C01810=1059.024,240.008,407.416,172.728,33.763,156.284
C01811=1059.018,239.759,407.444,172.726,33.759,156.283
C01812=1059.012,239.511,407.472,172.723,33.755,156.282
C01813=1059.006,239.263,407.499,172.721,33.752,156.282
C01814=1059.000,239.014,407.528,172.719,33.748,156.281
C01815=1058.993,238.765,407.555,172.717,33.744,156.280
C01816=1058.987,238.517,407.582,172.714,33.740,156.279
C01817=1058.981,238.269,407.610,172.712,33.737,156.279
C01818=1058.975,238.020,407.638,172.709,33.733,156.278
C01819=1058.969,237.772,407.665,172.707,33.729,156.277
C01820=1058.962,237.523,407.692,172.705,33.725,156.276
C01821=1058.956,237.275,407.720,172.703,33.721,156.276
C01822=1058.950,237.027,407.748,172.701,33.718,156.275
C01823=1058.944,236.778,407.775,172.699,33.714,156.274
C01824=1058.938,236.530,407.802,172.696,33.710,156.274
C01825=1058.932,236.297,407.829,172.694,33.707,156.273
C01826=1058.926,236.065,407.854,172.691,33.703,156.272
C01827=1058.920,235.833,407.879,172.689,33.700,156.272
C01828=1058.915,235.599,407.906,172.687,33.696,156.271
C01829=1058.909,235.367,407.931,172.685,33.692,156.270
C01830=1058.903,235.135,407.957,172.683,33.689,156.270
C01831=1058.897,234.902,407.983,172.681,33.685,156.269
C01832=1058.892,234.670,408.008,172.679,33.681,156.268
C01833=1058.885,234.421,408.036,172.677,33.678,156.267
C01834=1058.880,234.173,408.063,172.675,33.674,156.267
C01835=1058.873,233.924,408.090,172.673,33.670,156.266
C01836=1058.867,233.676,408.117,172.671,33.666,156.265
C01837=1058.861,233.427,408.145,172.668,33.663,156.265
C01838=1058.855,233.180,408.173,172.666,33.659,156.264
C01839=1058.849,232.930,408.200,172.664,33.655,156.263
C01840=1058.843,232.683,408.227,172.661,33.651,156.262
C01841=1058.836,232.434,408.254,172.659,33.647,156.262
C01842=1058.830,232.185,408.281,172.657,33.644,156.261
C01843=1058.824,231.937,408.309,172.655,33.639,156.260
C01844=1058.818,231.688,408.335,172.653,33.636,156.259
C01845=1058.811,231.440,408.363,172.651,33.632,156.259
C01846=1058.806,231.192,408.390,172.649,33.629,156.258
C01847=1058.800,230.943,408.418,172.647,33.624,156.257
C01848=1058.794,230.695,408.445,172.644,33.621,156.256
C01849=1058.787,230.445,408.472,172.641,33.617,156.256
C01850=1058.781,230.198,408.499,172.639,33.613,156.255
C01851=1058.775,229.949,408.526,172.637,33.609,156.254
C01852=1058.769,229.701,408.553,172.635,33.605,156.254
C01853=1058.763,229.452,408.580,172.633,33.601,156.253
C01854=1058.757,229.204,408.607,172.631,33.598,156.252
C01855=1058.750,228.954,408.634,172.629,33.594,156.251
C01856=1058.744,228.707,408.661,172.627,33.590,156.251
C01857=1058.737,228.458,408.688,172.625,33.587,156.250
C01858=1058.731,228.210,408.714,172.623,33.582,156.249
C01859=1058.725,227.961,408.742,172.620,33.579,156.248
C01860=1058.719,227.713,408.769,172.617,33.575,156.248
C01861=1058.713,227.464,408.795,172.615,33.571,156.247
C01862=1058.707,227.215,408.822,172.613,33.567,156.246
C01863=1058.700,226.967,408.848,172.611,33.564,156.246
C01864=1058.694,226.719,408.876,172.609,33.560,156.245
C01865=1058.688,226.471,408.903,172.607,33.556,156.244
C01866=1058.681,226.221,408.930,172.605,33.552,156.243
C01867=1058.676,225.973,408.957,172.603,33.548,156.243
C01868=1058.670,225.725,408.983,172.601,33.545,156.242
C01869=1058.663,225.476,409.010,172.599,33.540,156.241
C01870=1058.657,225.228,409.037,172.597,33.537,156.241
C01871=1058.650,224.979,409.064,172.595,33.533,156.240
C01872=1058.645,224.731,409.091,172.592,33.529,156.239
C01873=1058.639,224.483,409.117,172.590,33.525,156.238
C01874=1058.632,224.233,409.144,172.588,33.522,156.238
C01875=1058.626,223.985,409.170,172.586,33.517,156.237
C01876=1058.620,223.737,409.197,172.584,33.514,156.236
C01877=1058.614,223.488,409.224,172.582,33.510,156.235
C01878=1058.608,223.240,409.251,172.580,33.506,156.235
C01879=1058.602,222.991,409.277,172.578,33.502,156.234
C01880=1058.595,222.743,409.304,172.576,33.499,156.233
C01881=1058.590,222.506,409.330,172.574,33.495,156.233
C01882=1058.584,222.270,409.354,172.572,33.491,156.232
C01883=1058.578,222.033,409.380,172.570,33.488,156.231
C01884=1058.572,221.797,409.405,172.568,33.484,156.230
C01885=1058.566,221.561,409.430,172.565,33.480,156.230
C01886=1058.561,221.324,409.456,172.563,33.476,156.229
C01887=1058.555,221.088,409.481,172.561,33.472,156.228
C01888=1058.549,220.852,409.507,172.559,33.469,156.228
C01889=1058.543,220.603,409.532,172.557,33.465,156.227
C01890=1058.537,220.354,409.559,172.555,33.461,156.226
C01891=1058.530,220.106,409.585,172.553,33.458,156.225
C01892=1058.524,219.857,409.612,172.551,33.453,156.225
C01893=1058.517,219.609,409.638,172.549,33.450,156.224
C01894=1058.511,219.360,409.665,172.547,33.446,156.223
C01895=1058.505,219.112,409.691,172.545,33.442,156.222
C01896=1058.499,218.863,409.717,172.543,33.438,156.222
C01897=1058.493,218.614,409.744,172.541,33.435,156.221
C01898=1058.486,218.366,409.770,172.539,33.430,156.220
C01899=1058.481,218.118,409.797,172.537,33.427,156.220
C01900=1058.474,217.868,409.823,172.535,33.423,156.219
C01901=1058.468,217.620,409.849,172.532,33.419,156.218
C01902=1058.462,217.372,409.875,172.530,33.415,156.217
C01903=1058.456,217.124,409.902,172.528,33.411,156.217
C01904=1058.449,216.874,409.928,172.526,33.407,156.216
C01905=1058.443,216.626,409.954,172.524,33.404,156.215
C01906=1058.437,216.378,409.980,172.522,33.400,156.215
C01907=1058.431,216.129,410.007,172.520,33.396,156.214
C01908=1058.424,215.880,410.033,172.519,33.392,156.213
C01909=1058.418,215.632,410.059,172.517,33.388,156.212
C01910=1058.412,215.384,410.085,172.515,33.384,156.212
C01911=1058.406,215.135,410.111,172.513,33.380,156.211
C01912=1058.400,214.887,410.137,172.511,33.376,156.210
C01913=1058.394,214.637,410.164,172.509,33.373,156.209
C01914=1058.387,214.389,410.190,172.507,33.368,156.209
C01915=1058.382,214.141,410.216,172.505,33.365,156.208
C01916=1058.375,213.892,410.242,172.503,33.361,156.207
C01917=1058.370,213.644,410.268,172.500,33.357,156.206
C01918=1058.363,213.395,410.294,172.498,33.353,156.206
C01919=1058.358,213.147,410.320,172.496,33.349,156.205
C01920=1058.350,212.898,410.347,172.494,33.345,156.204
C01921=1058.345,212.649,410.373,172.492,33.341,156.203
C01922=1058.338,212.401,410.399,172.490,33.337,156.203
C01923=1058.333,212.152,410.425,172.488,33.334,156.202
C01924=1058.327,211.904,410.451,172.486,33.329,156.201
C01925=1058.320,211.655,410.476,172.485,33.326,156.200
C01926=1058.314,211.405,410.502,172.483,33.321,156.200
C01927=1058.308,211.157,410.528,172.481,33.318,156.199
C01928=1058.302,210.909,410.554,172.479,33.313,156.198
C01929=1058.296,210.660,410.580,172.477,33.310,156.197
C01930=1058.290,210.412,410.606,172.475,33.306,156.197
C01931=1058.283,210.164,410.632,172.473,33.302,156.196
C01932=1058.277,209.915,410.657,172.471,33.298,156.195
C01933=1058.271,209.666,410.683,172.469,33.294,156.194
C01934=1058.265,209.418,410.709,172.467,33.290,156.194
C01935=1058.258,209.168,410.735,172.465,33.287,156.193
C01936=1058.252,208.920,410.761,172.463,33.282,156.192
C01937=1058.246,208.686,410.785,172.461,33.279,156.192
C01938=1058.241,208.453,410.809,172.459,33.275,156.191
C01939=1058.234,208.219,410.833,172.457,33.271,156.190
C01940=1058.229,207.985,410.857,172.455,33.268,156.190
C01941=1058.223,207.751,410.881,172.454,33.264,156.189
C01942=1058.217,207.517,410.906,172.452,33.260,156.188
C01943=1058.212,207.283,410.930,172.450,33.257,156.187
C01944=1058.206,207.049,410.954,172.448,33.253,156.187
C01945=1058.180,205.999,411.059,172.259,33.165,156.176
C01946=1058.174,205.751,411.084,172.256,33.162,156.175
C01947=1058.169,205.502,411.108,172.254,33.159,156.175
C01948=1058.163,205.253,411.133,172.252,33.156,156.174
C01949=1058.157,205.005,411.157,172.249,33.153,156.173
C01950=1058.151,204.756,411.182,172.247,33.150,156.173
C01951=1058.145,204.507,411.207,172.245,33.147,156.172
C01952=1058.139,204.259,411.232,172.242,33.144,156.172
C01953=1058.133,204.010,411.257,172.240,33.140,156.171
C01954=1058.128,203.761,411.281,172.238,33.138,156.171
C01955=1058.122,203.512,411.306,172.235,33.135,156.170
C01956=1058.116,203.263,411.331,172.233,33.132,156.170
C01957=1058.110,203.015,411.355,172.231,33.128,156.169
C01958=1058.104,202.766,411.379,172.228,33.125,156.169
C01959=1058.098,202.518,411.404,172.225,33.122,156.168
C01960=1058.092,202.268,411.429,172.223,33.120,156.168
C01961=1058.087,202.020,411.453,172.220,33.116,156.167
C01962=1058.081,201.771,411.479,172.218,33.113,156.166
C01963=1058.074,201.522,411.503,172.216,33.110,156.166
C01964=1058.069,201.274,411.527,172.213,33.107,156.165
C01965=1058.062,201.025,411.551,172.211,33.104,156.165
C01966=1058.057,200.777,411.576,172.209,33.101,156.164
C01967=1058.050,200.528,411.600,172.207,33.099,156.164
C01968=1058.044,200.278,411.625,172.204,33.095,156.163
C01969=1058.039,200.030,411.649,172.202,33.093,156.163
C01970=1058.032,199.781,411.673,172.200,33.090,156.162
C01971=1058.026,199.533,411.698,172.197,33.087,156.162
C01972=1058.020,199.284,411.722,172.195,33.084,156.161
C01973=1058.015,199.035,411.746,172.193,33.081,156.161
C01974=1058.008,198.786,411.770,172.190,33.078,156.160
C01975=1058.003,198.538,411.794,172.188,33.075,156.160
C01976=1057.996,198.289,411.818,172.186,33.072,156.159
C01977=1057.991,198.040,411.843,172.184,33.069,156.159
C01978=1057.984,197.792,411.868,172.181,33.066,156.158
C01979=1057.978,197.543,411.892,172.179,33.063,156.158
C01980=1057.973,197.294,411.916,172.177,33.061,156.157
C01981=1057.966,197.045,411.940,172.174,33.057,156.157
C01982=1057.961,196.796,411.965,172.172,33.054,156.156
C01983=1057.955,196.548,411.988,172.170,33.052,156.156
C01984=1057.949,196.299,412.013,172.168,33.048,156.155
C01985=1057.943,196.051,412.036,172.166,33.046,156.155
C01986=1057.937,195.801,412.061,172.164,33.043,156.154
C01987=1057.931,195.553,412.085,172.162,33.040,156.154
C01988=1057.925,195.304,412.109,172.160,33.037,156.153
C01989=1057.919,195.055,412.133,172.157,33.034,156.153
C01990=1057.913,194.806,412.158,172.155,33.031,156.152
C01991=1057.907,194.558,412.181,172.153,33.028,156.152
C01992=1057.901,194.309,412.206,172.151,33.025,156.151
C01993=1057.895,194.060,412.230,172.148,33.022,156.151
C01994=1057.890,193.812,412.254,172.146,33.019,156.150
C01995=1057.883,193.562,412.277,172.144,33.017,156.150
C01996=1057.878,193.314,412.301,172.142,33.014,156.149
C01997=1057.871,193.065,412.325,172.140,33.010,156.149
C01998=1057.866,192.816,412.350,172.137,33.008,156.148
C01999=1057.860,192.568,412.373,172.135,33.005,156.148
C02000=1057.854,192.318,412.398,172.133,33.002,156.147
C02001=1057.848,192.070,412.422,172.131,32.999,156.147
C02002=1057.843,191.821,412.445,172.128,32.996,156.146
C02003=1057.836,191.572,412.469,172.126,32.993,156.146
C02004=1057.831,191.323,412.493,172.124,32.990,156.145
C02005=1057.824,191.074,412.518,172.122,32.987,156.145
C02006=1057.819,190.791,412.544,172.119,32.984,156.144
C02007=1057.812,190.507,412.572,172.117,32.980,156.143
C02008=1057.805,190.223,412.599,172.114,32.977,156.143
C02009=1057.799,189.940,412.627,172.112,32.974,156.142
C02010=1057.792,189.691,412.651,172.110,32.971,156.142
C02011=1057.787,189.442,412.674,172.107,32.968,156.141
C02012=1057.781,189.193,412.698,172.105,32.965,156.141
C02013=1057.774,188.944,412.722,172.103,32.963,156.140
C02014=1057.769,188.695,412.745,172.101,32.959,156.140
C02015=1057.763,188.447,412.769,172.099,32.957,156.139
C02016=1057.758,188.198,412.793,172.096,32.954,156.139
C02017=1057.752,187.949,412.817,172.094,32.951,156.138
C02018=1057.746,187.700,412.841,172.092,32.948,156.138
C02019=1057.740,187.452,412.864,172.090,32.945,156.137
C02020=1057.735,187.203,412.887,172.088,32.942,156.137
C02021=1057.729,186.954,412.912,172.086,32.939,156.136
C02022=1057.723,186.705,412.936,172.083,32.936,156.136
C02023=1057.718,186.456,412.959,172.081,32.933,156.135
C02024=1057.712,186.208,412.983,172.079,32.931,156.135
C02025=1057.706,185.958,413.007,172.077,32.928,156.134
C02026=1057.700,185.710,413.030,172.075,32.925,156.134
C02027=1057.694,185.461,413.054,172.073,32.922,156.133
C02028=1057.689,185.212,413.078,172.071,32.919,156.133
C02029=1057.683,184.964,413.101,172.068,32.916,156.132
C02030=1057.677,184.714,413.125,172.066,32.913,156.132
C02031=1057.671,184.466,413.149,172.064,32.910,156.131
C02032=1057.666,184.217,413.172,172.062,32.908,156.131
C02033=1057.660,183.969,413.196,172.060,32.905,156.130
C02034=1057.653,183.719,413.219,172.058,32.902,156.130
C02035=1057.647,183.470,413.242,172.055,32.899,156.129
C02036=1057.641,183.222,413.265,172.053,32.897,156.129
C02037=1057.635,182.972,413.289,172.051,32.894,156.128
C02038=1057.629,182.724,413.312,172.049,32.891,156.128
C02039=1057.623,182.475,413.335,172.047,32.889,156.128
C02040=1057.618,182.226,413.358,172.045,32.886,156.127
C02041=1057.610,181.977,413.382,172.042,32.883,156.127
C02042=1057.604,181.729,413.405,172.040,32.880,156.126
C02043=1057.599,181.480,413.428,172.038,32.878,156.126
C02044=1057.593,181.231,413.451,172.036,32.875,156.125
C02045=1057.586,180.982,413.475,172.034,32.872,156.125
C02046=1057.581,180.733,413.498,172.032,32.869,156.124
C02047=1057.575,180.485,413.521,172.030,32.867,156.124
C02048=1057.569,180.236,413.544,172.027,32.864,156.123
C02049=1057.563,179.986,413.567,172.025,32.862,156.123
C02050=1057.557,179.737,413.590,172.023,32.858,156.122
C02051=1057.550,179.489,413.613,172.021,32.856,156.122
C02052=1057.544,179.240,413.636,172.019,32.853,156.122
C02053=1057.539,178.991,413.659,172.017,32.851,156.121
C02054=1057.532,178.742,413.683,172.015,32.848,156.121
C02055=1057.526,178.494,413.706,172.013,32.845,156.120
C02056=1057.520,178.245,413.729,172.011,32.842,156.120
C02057=1057.515,177.996,413.752,172.009,32.840,156.119
C02058=1057.509,177.747,413.775,172.007,32.837,156.119
C02059=1057.502,177.498,413.798,172.005,32.834,156.118
C02060=1057.496,177.249,413.822,172.003,32.831,156.118
C02061=1057.490,177.000,413.845,172.001,32.829,156.117
C02062=1057.484,176.752,413.867,171.999,32.826,156.117
C02063=1057.479,176.503,413.890,171.997,32.823,156.116
C02064=1057.473,176.254,413.913,171.995,32.821,156.116
C02065=1057.467,176.005,413.936,171.993,32.818,156.116
C02066=1057.461,175.756,413.959,171.990,32.815,156.115
C02067=1057.454,175.507,413.982,171.988,32.812,156.115
C02068=1057.448,175.258,414.006,171.986,32.810,156.114
C02069=1057.443,175.009,414.029,171.984,32.807,156.114
C02070=1057.436,174.725,414.054,171.982,32.804,156.113
C02071=1057.429,174.441,414.081,171.979,32.801,156.113
C02072=1057.422,174.156,414.107,171.977,32.798,156.112
C02073=1057.416,173.872,414.133,171.975,32.795,156.112
C02074=1057.410,173.623,414.156,171.973,32.792,156.111
C02075=1057.404,173.374,414.178,171.971,32.789,156.111
C02076=1057.398,173.125,414.201,171.968,32.786,156.110
C02077=1057.393,172.876,414.224,171.966,32.784,156.110
C02078=1057.386,172.628,414.247,171.964,32.781,156.109
C02079=1057.380,172.379,414.270,171.962,32.778,156.109
C02080=1057.375,172.130,414.293,171.960,32.776,156.108
C02081=1057.369,171.881,414.316,171.958,32.773,156.108
C02082=1057.363,171.632,414.339,171.956,32.770,156.108
C02083=1057.357,171.384,414.361,171.954,32.768,156.107
C02084=1057.351,171.135,414.384,171.952,32.765,156.107
C02085=1057.345,170.886,414.407,171.950,32.762,156.106
C02086=1057.340,170.637,414.430,171.948,32.760,156.106
C02087=1057.334,170.388,414.453,171.946,32.757,156.105
C02088=1057.327,170.139,414.475,171.944,32.754,156.105
C02089=1057.322,169.891,414.498,171.942,32.751,156.104
C02090=1057.316,169.641,414.520,171.940,32.749,156.104
C02091=1057.311,169.392,414.543,171.939,32.746,156.103
C02092=1057.305,169.143,414.566,171.937,32.744,156.103
C02093=1057.298,168.895,414.588,171.935,32.740,156.102
C02094=1057.293,168.646,414.611,171.933,32.738,156.102
C02095=1057.287,168.397,414.634,171.931,32.735,156.102
C02096=1057.281,168.147,414.657,171.929,32.733,156.101
C02097=1057.275,167.899,414.679,171.927,32.730,156.101
C02098=1057.269,167.650,414.702,171.925,32.727,156.100
C02099=1057.264,167.402,414.724,171.923,32.724,156.100
C02100=1057.258,167.153,414.747,171.921,32.722,156.099
C02101=1057.252,166.904,414.769,171.919,32.719,156.099
C02102=1057.246,166.655,414.792,171.917,32.716,156.098
C02103=1057.241,166.406,414.815,171.915,32.713,156.098
C02104=1057.235,166.157,414.838,171.913,32.711,156.097
C02105=1057.229,165.908,414.859,171.911,32.708,156.097
C02106=1057.223,165.659,414.882,171.909,32.706,156.097
C02107=1057.217,165.410,414.905,171.907,32.702,156.096
C02108=1057.213,165.161,414.927,171.905,32.700,156.096
C02109=1057.206,164.913,414.950,171.903,32.697,156.095
C02110=1057.200,164.664,414.973,171.901,32.695,156.095
C02111=1057.195,164.414,414.995,171.899,32.692,156.094
C02112=1057.189,164.165,415.018,171.897,32.689,156.094
C02113=1057.183,163.917,415.040,171.895,32.686,156.093
C02114=1057.177,163.667,415.062,171.893,32.684,156.093
C02115=1057.172,163.419,415.085,171.891,32.681,156.092
C02116=1057.166,163.170,415.108,171.889,32.678,156.092
C02117=1057.160,162.921,415.129,171.887,32.675,156.091
C02118=1057.155,162.672,415.152,171.885,32.673,156.091
C02119=1057.149,162.422,415.175,171.884,32.670,156.091
C02120=1057.143,162.175,415.197,171.882,32.668,156.090
C02121=1057.138,161.926,415.220,171.880,32.665,156.090
C02122=1057.132,161.676,415.242,171.878,32.662,156.089
C02123=1057.126,161.427,415.265,171.876,32.659,156.089
C02124=1057.120,161.178,415.286,171.874,32.657,156.088
C02125=1057.115,160.930,415.309,171.872,32.654,156.088
C02126=1057.109,160.681,415.331,171.870,32.651,156.087
C02127=1057.103,160.432,415.354,171.868,32.648,156.087
C02128=1057.097,160.182,415.375,171.866,32.646,156.087
C02129=1057.091,159.934,415.397,171.864,32.643,156.086
C02130=1057.085,159.684,415.420,171.862,32.641,156.086
C02131=1057.079,159.435,415.441,171.860,32.638,156.085
C02132=1057.074,159.187,415.464,171.858,32.636,156.085
C02133=1057.068,158.938,415.486,171.856,32.633,156.084
C02134=1057.061,158.653,415.511,171.854,32.630,156.084
C02135=1057.054,158.368,415.536,171.852,32.627,156.083
C02136=1057.047,158.084,415.561,171.849,32.624,156.083
C02137=1057.040,157.799,415.586,171.847,32.621,156.082
C02138=1057.034,157.550,415.609,171.845,32.619,156.082
C02139=1057.029,157.302,415.630,171.843,32.616,156.082
C02140=1057.023,157.052,415.652,171.841,32.614,156.081
C02141=1057.017,156.804,415.675,171.839,32.611,156.081
C02142=1057.011,156.554,415.697,171.837,32.608,156.080
C02143=1057.005,156.305,415.718,171.836,32.606,156.080
C02144=1056.999,156.057,415.741,171.835,32.603,156.079
C02145=1056.993,155.808,415.763,171.833,32.601,156.079
C02146=1056.987,155.559,415.784,171.831,32.598,156.079
C02147=1056.981,155.310,415.807,171.829,32.595,156.078
C02148=1056.976,155.061,415.828,171.827,32.593,156.078
C02149=1056.970,154.812,415.850,171.825,32.590,156.077
C02150=1056.963,154.563,415.872,171.823,32.588,156.077
C02151=1056.958,154.314,415.895,171.821,32.585,156.076
C02152=1056.952,154.065,415.916,171.819,32.583,156.076
C02153=1056.946,153.816,415.938,171.817,32.580,156.076
C02154=1056.940,153.567,415.959,171.815,32.577,156.075
C02155=1056.934,153.318,415.981,171.813,32.575,156.075
C02156=1056.928,153.069,416.004,171.811,32.572,156.074
C02157=1056.922,152.820,416.025,171.809,32.570,156.074
C02158=1056.916,152.571,416.047,171.807,32.567,156.073
C02159=1056.910,152.322,416.068,171.805,32.564,156.073
C02160=1056.904,152.073,416.090,171.804,32.562,156.072
C02161=1056.898,151.824,416.111,171.802,32.559,156.072
C02162=1056.893,151.575,416.133,171.800,32.557,156.072
C02163=1056.887,151.325,416.155,171.798,32.554,156.071
C02164=1056.881,151.078,416.177,171.796,32.552,156.071
C02165=1056.875,150.828,416.199,171.795,32.549,156.070
C02166=1056.869,150.579,416.220,171.793,32.546,156.070
C02167=1056.863,150.331,416.242,171.791,32.544,156.069
C02168=1056.858,150.081,416.264,171.789,32.541,156.069
C02169=1056.851,149.832,416.285,171.787,32.539,156.069
C02170=1056.846,149.583,416.307,171.785,32.536,156.068
C02171=1056.840,149.334,416.328,171.784,32.533,156.068
C02172=1056.833,149.085,416.350,171.782,32.531,156.067
C02173=1056.828,148.836,416.371,171.780,32.528,156.067
C02174=1056.822,148.587,416.393,171.778,32.526,156.066
C02175=1056.816,148.338,416.415,171.776,32.523,156.066
C02176=1056.810,148.090,416.436,171.774,32.521,156.066
C02177=1056.804,147.840,416.457,171.772,32.518,156.065
C02178=1056.798,147.591,416.480,171.770,32.516,156.065
C02179=1056.792,147.343,416.500,171.768,32.513,156.064
C02180=1056.786,147.093,416.522,171.766,32.511,156.064
C02181=1056.780,146.844,416.544,171.765,32.508,156.064
C02182=1056.774,146.596,416.565,171.763,32.506,156.063
C02183=1056.768,146.347,416.587,171.761,32.503,156.063
C02184=1056.762,146.097,416.607,171.759,32.500,156.062
C02185=1056.757,145.848,416.629,171.758,32.498,156.062
C02186=1056.751,145.599,416.650,171.756,32.496,156.062
C02187=1056.744,145.350,416.672,171.754,32.493,156.061
C02188=1056.739,145.101,416.693,171.752,32.491,156.061
C02189=1056.733,144.852,416.715,171.750,32.488,156.060
C02190=1056.726,144.603,416.737,171.748,32.485,156.060
C02191=1056.721,144.354,416.758,171.747,32.483,156.059
C02192=1056.715,144.105,416.779,171.745,32.480,156.059
C02193=1056.709,143.856,416.799,171.743,32.478,156.059
C02194=1056.703,143.607,416.821,171.741,32.476,156.058
C02195=1056.696,143.358,416.843,171.739,32.473,156.058
C02196=1056.691,143.109,416.864,171.737,32.470,156.057
C02197=1056.685,142.860,416.885,171.735,32.468,156.057
C02198=1056.678,142.575,416.910,171.733,32.465,156.056
C02199=1056.672,142.290,416.934,171.731,32.462,156.056
C02200=1056.665,142.005,416.957,171.729,32.459,156.055
C02201=1056.658,141.720,416.982,171.727,32.456,156.055
C02202=1056.653,141.472,417.004,171.725,32.454,156.055
C02203=1056.646,141.222,417.025,171.724,32.451,156.054
C02204=1056.640,140.973,417.046,171.722,32.448,156.054
C02205=1056.634,140.724,417.067,171.720,32.446,156.053
C02206=1056.628,140.475,417.089,171.719,32.444,156.053
C02207=1056.623,140.226,417.109,171.717,32.441,156.053
C02208=1056.617,139.977,417.131,171.715,32.439,156.052
C02209=1056.611,139.728,417.152,171.713,32.436,156.052
C02210=1056.605,139.478,417.173,171.711,32.434,156.051
C02211=1056.599,139.230,417.194,171.709,32.431,156.051
C02212=1056.593,138.981,417.215,171.707,32.428,156.050
C02213=1056.588,138.732,417.236,171.706,32.426,156.050
C02214=1056.581,138.483,417.257,171.704,32.424,156.050
C02215=1056.575,138.234,417.277,171.702,32.421,156.049
C02216=1056.569,137.985,417.299,171.700,32.419,156.049
C02217=1056.563,137.735,417.321,171.698,32.416,156.048
C02218=1056.557,137.487,417.341,171.696,32.413,156.048
C02219=1056.551,137.237,417.362,171.695,32.411,156.048
C02220=1056.546,136.988,417.383,171.693,32.409,156.047
C02221=1056.539,136.739,417.404,171.692,32.406,156.047
C02222=1056.533,136.490,417.424,171.690,32.404,156.046
C02223=1056.527,136.241,417.446,171.688,32.401,156.046
C02224=1056.521,135.992,417.466,171.686,32.398,156.046
C02225=1056.515,135.743,417.488,171.684,32.396,156.045
C02226=1056.510,135.494,417.508,171.683,32.394,156.045
C02227=1056.503,135.245,417.529,171.681,32.391,156.044
C02228=1056.498,134.996,417.550,171.679,32.389,156.044
C02229=1056.492,134.747,417.571,171.677,32.386,156.043
C02230=1056.486,134.498,417.591,171.675,32.384,156.043
C02231=1056.479,134.249,417.613,171.673,32.381,156.043
C02232=1056.474,134.000,417.634,171.672,32.379,156.042
C02233=1056.468,133.751,417.654,171.670,32.376,156.042
C02234=1056.462,133.502,417.675,171.668,32.374,156.041
C02235=1056.457,133.252,417.696,171.666,32.371,156.041
C02236=1056.450,133.004,417.717,171.664,32.369,156.041
C02237=1056.445,132.754,417.737,171.664,32.367,156.040
C02238=1056.438,132.506,417.758,171.662,32.364,156.040
C02239=1056.432,132.256,417.779,171.660,32.361,156.039
C02240=1056.427,132.007,417.799,171.658,32.359,156.039
C02241=1056.420,131.758,417.820,171.656,32.356,156.039
C02242=1056.415,131.509,417.841,171.654,32.354,156.038
C02243=1056.408,131.260,417.861,171.653,32.352,156.038
C02244=1056.403,131.011,417.883,171.651,32.349,156.037
C02245=1056.396,130.762,417.903,171.649,32.347,156.037
C02246=1056.390,130.513,417.923,171.647,32.344,156.037
C02247=1056.384,130.264,417.945,171.645,32.342,156.036
C02248=1056.378,130.015,417.965,171.644,32.340,156.036
C02249=1056.372,129.765,417.985,171.642,32.337,156.035
C02250=1056.366,129.516,418.005,171.640,32.335,156.035
C02251=1056.359,129.267,418.026,171.638,32.332,156.035
C02252=1056.353,129.019,418.046,171.636,32.330,156.034
C02253=1056.348,128.769,418.067,171.635,32.327,156.034
C02254=1056.342,128.520,418.087,171.634,32.325,156.033
C02255=1056.336,128.271,418.109,171.632,32.323,156.033
C02256=1056.329,128.022,418.129,171.630,32.320,156.033
C02257=1056.323,127.773,418.149,171.628,32.318,156.032
C02258=1056.318,127.523,418.170,171.626,32.315,156.032
C02259=1056.312,127.274,418.190,171.625,32.313,156.032
C02260=1056.306,127.026,418.210,171.623,32.311,156.031
C02261=1056.299,126.776,418.231,171.621,32.308,156.031
C02262=1056.292,126.492,418.254,171.619,32.305,156.030
C02263=1056.285,126.207,418.278,171.617,32.303,156.030
C02264=1056.279,125.922,418.301,171.615,32.300,156.029
C02265=1056.272,125.636,418.324,171.613,32.297,156.029
C02266=1056.266,125.388,418.345,171.611,32.295,156.029
C02267=1056.259,125.138,418.365,171.609,32.292,156.028
C02268=1056.254,124.889,418.385,171.608,32.290,156.028
C02269=1056.248,124.640,418.405,171.607,32.287,156.027
C02270=1056.241,124.391,418.426,171.605,32.285,156.027
C02271=1056.236,124.142,418.446,171.603,32.282,156.027
C02272=1056.230,123.893,418.466,171.601,32.280,156.026
C02273=1056.224,123.643,418.487,171.600,32.277,156.026
C02274=1056.218,123.395,418.507,171.598,32.275,156.025
C02275=1056.212,123.145,418.527,171.596,32.273,156.025
C02276=1056.206,122.896,418.547,171.594,32.270,156.025
C02277=1056.200,122.647,418.567,171.592,32.268,156.024
C02278=1056.194,122.398,418.588,171.591,32.265,156.024
C02279=1056.188,122.148,418.608,171.589,32.263,156.023
C02280=1056.182,121.900,418.628,171.587,32.260,156.023
C02281=1056.177,121.651,418.649,171.585,32.258,156.023
C02282=1056.171,121.402,418.669,171.585,32.256,156.022
C02283=1056.164,121.152,418.689,171.583,32.253,156.022
C02284=1056.158,120.903,418.709,171.581,32.250,156.021
C02285=1056.153,120.654,418.730,171.579,32.248,156.021
C02286=1056.146,120.405,418.750,171.577,32.246,156.021
C02287=1056.140,120.156,418.770,171.576,32.243,156.020
C02288=1056.134,119.907,418.790,171.574,32.241,156.020
C02289=1056.129,119.658,418.810,171.572,32.238,156.019
C02290=1056.122,119.408,418.831,171.570,32.236,156.019
C02291=1056.116,119.160,418.851,171.569,32.234,156.019
C02292=1056.111,118.911,418.871,171.567,32.231,156.018
C02293=1056.105,118.662,418.891,171.565,32.228,156.018
C02294=1056.099,118.412,418.910,171.563,32.226,156.017
C02295=1056.093,118.163,418.931,171.562,32.224,156.017
C02296=1056.088,117.914,418.951,171.561,32.221,156.017
C02297=1056.082,117.665,418.971,171.559,32.218,156.016
C02298=1056.076,117.416,418.991,171.557,32.216,156.016
C02299=1056.070,117.167,419.011,171.556,32.214,156.015
C02300=1056.064,116.917,419.032,171.554,32.211,156.015
C02301=1056.058,116.668,419.051,171.552,32.209,156.015
C02302=1056.052,116.419,419.071,171.550,32.206,156.014
C02303=1056.046,116.170,419.091,171.549,32.204,156.014
C02304=1056.041,115.921,419.112,171.547,32.202,156.013
C02305=1056.034,115.672,419.132,171.545,32.199,156.013
C02306=1056.028,115.422,419.151,171.543,32.196,156.013
C02307=1056.022,115.173,419.171,171.542,32.194,156.012
C02308=1056.016,114.925,419.191,171.540,32.192,156.012
C02309=1056.011,114.676,419.212,171.538,32.189,156.011
C02310=1056.006,114.426,419.231,171.538,32.187,156.011
C02311=1056.000,114.177,419.251,171.536,32.184,156.011
C02312=1055.993,113.928,419.271,171.534,32.181,156.010
C02313=1055.987,113.679,419.291,171.532,32.179,156.010
C02314=1055.981,113.430,419.311,171.531,32.177,156.009
C02315=1055.975,113.181,419.330,171.529,32.174,156.009
C02316=1055.969,112.932,419.350,171.527,32.172,156.009
C02317=1055.963,112.682,419.370,171.525,32.169,156.008
C02318=1055.957,112.433,419.390,171.524,32.167,156.008
C02319=1055.951,112.184,419.410,171.522,32.165,156.008
C02320=1055.945,111.935,419.429,171.520,32.162,156.007
C02321=1055.939,111.686,419.449,171.518,32.160,156.007
C02322=1055.933,111.437,419.469,171.517,32.158,156.006
C02323=1055.927,111.187,419.489,171.516,32.155,156.006
C02324=1055.921,110.938,419.509,171.514,32.153,156.006
C02325=1055.915,110.689,419.528,171.512,32.150,156.005
C02326=1055.908,110.404,419.551,171.510,32.147,156.005
C02327=1055.902,110.118,419.574,171.508,32.145,156.004
C02328=1055.895,109.833,419.596,171.506,32.142,156.004
C02329=1055.888,109.548,419.618,171.505,32.139,156.003
C02330=1055.882,109.300,419.637,171.503,32.137,156.003
C02331=1055.876,109.049,419.657,171.501,32.135,156.003
C02332=1055.870,108.801,419.677,171.499,32.132,156.002
C02333=1055.863,108.551,419.696,171.498,32.130,156.002
C02334=1055.857,108.303,419.716,171.496,32.128,156.002
C02335=1055.851,108.053,419.735,171.495,32.125,156.001
C02336=1055.845,107.804,419.755,171.493,32.123,156.001
C02337=1055.840,107.555,419.774,171.492,32.120,156.000
C02338=1055.833,107.305,419.794,171.490,32.118,156.000
C02339=1055.827,107.056,419.813,171.488,32.116,156.000
C02340=1055.821,106.807,419.833,171.486,32.113,155.999
C02341=1055.815,106.558,419.852,171.485,32.111,155.999
C02342=1055.809,106.309,419.872,171.483,32.109,155.998
C02343=1055.803,106.060,419.891,171.481,32.106,155.998
C02344=1055.797,105.811,419.911,171.480,32.103,155.998
C02345=1055.791,105.562,419.930,171.478,32.101,155.997
C02346=1055.785,105.312,419.949,171.476,32.099,155.997
C02347=1055.779,105.064,419.969,171.474,32.096,155.996
C02348=1055.774,104.814,419.989,171.474,32.094,155.996
C02349=1055.767,104.566,420.008,171.472,32.092,155.996
C02350=1055.761,104.316,420.027,171.470,32.089,155.995
C02351=1055.755,104.067,420.046,171.469,32.087,155.995
C02352=1055.749,103.817,420.067,171.467,32.084,155.995
C02353=1055.743,103.568,420.086,171.465,32.082,155.994
C02354=1055.737,103.319,420.105,171.463,32.080,155.994
C02355=1055.731,103.070,420.125,171.462,32.077,155.993
C02356=1055.725,102.821,420.144,171.460,32.075,155.993
C02357=1055.719,102.571,420.163,171.458,32.072,155.993
C02358=1055.713,102.322,420.183,171.457,32.070,155.992
C02359=1055.707,102.073,420.202,171.455,32.067,155.992
C02360=1055.701,101.824,420.221,171.454,32.065,155.992
C02361=1055.695,101.575,420.241,171.453,32.063,155.991
C02362=1055.690,101.325,420.260,171.451,32.060,155.991
C02363=1055.683,101.076,420.279,171.449,32.058,155.990
C02364=1055.678,100.827,420.298,171.447,32.055,155.990
C02365=1055.672,100.578,420.318,171.446,32.053,155.990
C02366=1055.665,100.329,420.337,171.444,32.051,155.989
C02367=1055.659,100.080,420.356,171.442,32.048,155.989
C02368=1055.654,99.830,420.375,171.441,32.046,155.988
C02369=1055.647,99.581,420.394,171.439,32.044,155.988
C02370=1055.641,99.332,420.414,171.437,32.041,155.988
C02371=1055.635,99.083,420.432,171.435,32.039,155.987
C02372=1055.629,98.834,420.452,171.435,32.036,155.987
C02373=1055.623,98.585,420.470,171.433,32.034,155.987
C02374=1055.617,98.335,420.489,171.431,32.032,155.986
C02375=1055.611,98.086,420.508,171.430,32.029,155.986
C02376=1055.605,97.837,420.528,171.428,32.027,155.985
C02377=1055.598,97.588,420.547,171.426,32.025,155.985
C02378=1055.593,97.339,420.566,171.424,32.022,155.985
C02379=1055.586,97.089,420.585,171.423,32.020,155.984
C02380=1055.580,96.840,420.604,171.421,32.018,155.984
C02381=1055.575,96.591,420.623,171.419,32.015,155.984
C02382=1055.568,96.341,420.642,171.418,32.013,155.983
C02383=1055.563,96.092,420.661,171.417,32.011,155.983
C02384=1055.556,95.843,420.680,171.415,32.008,155.982
C02385=1055.551,95.593,420.699,171.414,32.006,155.982
C02386=1055.544,95.344,420.718,171.412,32.004,155.982
C02387=1055.538,95.096,420.738,171.410,32.001,155.981
C02388=1055.532,94.847,420.756,171.408,31.999,155.981
C02389=1055.527,94.598,420.775,171.407,31.996,155.981
C02390=1055.520,94.312,420.796,171.405,31.994,155.980
C02391=1055.512,94.027,420.818,171.403,31.991,155.980
C02392=1055.506,93.742,420.840,171.401,31.988,155.979
C02393=1055.499,93.457,420.861,171.399,31.986,155.979
C02394=1055.493,93.207,420.880,171.398,31.983,155.978
C02395=1055.487,92.958,420.899,171.397,31.981,155.978
C02396=1055.481,92.709,420.917,171.395,31.978,155.978
C02397=1055.475,92.460,420.937,171.393,31.976,155.977
C02398=1055.468,92.211,420.955,171.392,31.973,155.977
C02399=1055.463,91.961,420.975,171.390,31.971,155.977
C02400=1055.456,91.712,420.993,171.388,31.969,155.976
C02401=1055.451,91.463,421.012,171.387,31.967,155.976
C02402=1055.445,91.214,421.031,171.385,31.964,155.975
C02403=1055.439,90.965,421.050,171.383,31.961,155.975
C02404=1055.433,90.716,421.069,171.382,31.959,155.975
C02405=1055.427,90.466,421.088,171.381,31.957,155.974
C02406=1055.421,90.217,421.107,171.379,31.955,155.974
C02407=1055.414,89.967,421.124,171.377,31.952,155.974
C02408=1055.409,89.718,421.144,171.376,31.950,155.973
C02409=1055.402,89.469,421.162,171.374,31.948,155.973
C02410=1055.396,89.220,421.181,171.372,31.945,155.972
C02411=1055.390,88.971,421.199,171.371,31.943,155.972
C02412=1055.384,88.722,421.219,171.369,31.940,155.972
C02413=1055.378,88.472,421.236,171.367,31.938,155.971
C02414=1055.372,88.223,421.255,171.366,31.936,155.971
C02415=1055.365,87.974,421.274,171.364,31.934,155.971
C02416=1055.359,87.725,421.292,171.363,31.931,155.970
C02417=1055.353,87.475,421.312,171.361,31.929,155.970
C02418=1055.347,87.225,421.330,171.360,31.926,155.969
C02419=1055.341,86.977,421.348,171.358,31.924,155.969
C02420=1055.335,86.728,421.367,171.356,31.922,155.969
C02421=1055.329,86.479,421.386,171.355,31.920,155.968
C02422=1055.323,86.229,421.404,171.353,31.917,155.968
C02423=1055.317,85.980,421.422,171.351,31.915,155.968
C02424=1055.310,85.731,421.441,171.350,31.913,155.967
C02425=1055.304,85.482,421.459,171.348,31.910,155.967
C02426=1055.299,85.232,421.478,171.346,31.908,155.967
C02427=1055.293,84.983,421.496,171.346,31.905,155.966
C02428=1055.286,84.734,421.515,171.344,31.903,155.966
C02429=1055.280,84.484,421.533,171.342,31.901,155.965
C02430=1055.274,84.235,421.552,171.341,31.899,155.965
C02431=1055.269,83.986,421.571,171.339,31.896,155.965
C02432=1055.262,83.736,421.589,171.337,31.894,155.964
C02433=1055.256,83.487,421.607,171.336,31.891,155.964
C02434=1055.250,83.238,421.626,171.334,31.889,155.964
C02435=1055.244,82.989,421.643,171.332,31.887,155.963
C02436=1055.238,82.740,421.663,171.331,31.884,155.963
C02437=1055.232,82.491,421.681,171.330,31.882,155.962
C02438=1055.226,82.241,421.699,171.328,31.879,155.962
C02439=1055.219,81.992,421.718,171.327,31.878,155.962
C02440=1055.214,81.743,421.735,171.325,31.875,155.961
C02441=1055.208,81.493,421.755,171.323,31.873,155.961
C02442=1055.202,81.244,421.773,171.321,31.870,155.961
C02443=1055.196,80.994,421.791,171.320,31.868,155.960
C02444=1055.190,80.746,421.810,171.318,31.866,155.960
C02445=1055.184,80.496,421.827,171.316,31.863,155.959
C02446=1055.177,80.247,421.846,171.315,31.861,155.959
C02447=1055.173,79.998,421.864,171.313,31.858,155.959
C02448=1055.166,79.749,421.883,171.312,31.856,155.958
C02449=1055.160,79.499,421.901,171.311,31.854,155.958
C02450=1055.154,79.250,421.920,171.309,31.851,155.958
C02451=1055.148,79.001,421.938,171.307,31.849,155.957
C02452=1055.142,78.752,421.956,171.306,31.846,155.957
C02453=1055.135,78.503,421.974,171.304,31.844,155.957
C02454=1055.129,78.218,421.995,171.302,31.842,155.956
C02455=1055.122,77.932,422.016,171.300,31.839,155.956
C02456=1055.115,77.647,422.037,171.298,31.836,155.955
C02457=1055.108,77.361,422.058,171.297,31.834,155.955
C02458=1055.102,77.112,422.076,171.296,31.831,155.954
C02459=1055.096,76.864,422.093,171.294,31.829,155.954
C02460=1055.089,76.614,422.111,171.292,31.827,155.954
C02461=1055.083,76.364,422.129,171.291,31.825,155.953
C02462=1055.077,76.116,422.148,171.289,31.822,155.953
C02463=1055.071,75.866,422.166,171.287,31.820,155.953
C02464=1055.065,75.617,422.184,171.286,31.817,155.952
C02465=1055.059,75.367,422.202,171.284,31.815,155.952
C02466=1055.053,75.118,422.220,171.282,31.813,155.952
C02467=1055.047,74.869,422.238,171.282,31.811,155.951
C02468=1055.041,74.619,422.256,171.280,31.808,155.951
C02469=1055.035,74.370,422.274,171.278,31.806,155.951
C02470=1055.029,74.121,422.293,171.277,31.803,155.950
C02471=1055.023,73.871,422.310,171.275,31.801,155.950
C02472=1055.017,73.622,422.328,171.273,31.799,155.949
C02473=1055.010,73.373,422.346,171.272,31.797,155.949
C02474=1055.004,73.124,422.364,171.270,31.794,155.949
C02475=1054.998,72.875,422.382,171.268,31.792,155.948
C02476=1054.992,72.626,422.400,171.267,31.789,155.948
C02477=1054.986,72.376,422.418,171.266,31.787,155.948
C02478=1054.980,72.127,422.436,171.264,31.785,155.947
C02479=1054.974,71.877,422.454,171.263,31.783,155.947
C02480=1054.968,71.629,422.472,171.261,31.780,155.947
C02481=1054.962,71.379,422.490,171.259,31.778,155.946
C02482=1054.955,71.129,422.507,171.258,31.776,155.946
C02483=1054.950,70.880,422.525,171.256,31.773,155.945
C02484=1054.943,70.631,422.543,171.254,31.771,155.945
C02485=1054.937,70.381,422.561,171.253,31.769,155.945
C02486=1054.932,70.132,422.579,171.251,31.766,155.944
C02487=1054.926,69.883,422.597,171.250,31.764,155.944
C02488=1054.920,69.634,422.614,171.249,31.762,155.944
C02489=1054.913,69.385,422.632,171.247,31.760,155.943
C02490=1054.907,69.135,422.650,171.245,31.757,155.943
C02491=1054.901,68.886,422.668,171.244,31.755,155.943
C02492=1054.895,68.636,422.686,171.242,31.752,155.942
C02493=1054.889,68.388,422.703,171.240,31.750,155.942
C02494=1054.883,68.138,422.721,171.239,31.748,155.942
C02495=1054.876,67.889,422.739,171.237,31.746,155.941
C02496=1054.870,67.640,422.756,171.236,31.744,155.941
C02497=1054.864,67.390,422.774,171.235,31.741,155.940
C02498=1054.858,67.141,422.792,171.233,31.739,155.940
C02499=1054.852,66.891,422.810,171.231,31.736,155.940
C02500=1054.846,66.642,422.827,171.230,31.734,155.939
C02501=1054.840,66.393,422.845,171.228,31.732,155.939
C02502=1054.834,66.143,422.863,171.226,31.730,155.939
C02503=1054.828,65.895,422.880,171.224,31.727,155.938
C02504=1054.822,65.645,422.898,171.223,31.725,155.938
C02505=1054.816,65.396,422.915,171.221,31.723,155.938
C02506=1054.809,65.146,422.933,171.220,31.720,155.937
C02507=1054.803,64.897,422.950,171.219,31.718,155.937
C02508=1054.797,64.648,422.968,171.217,31.716,155.937
C02509=1054.791,64.398,422.985,171.215,31.714,155.936
C02510=1054.785,64.149,423.003,171.214,31.711,155.936
C02511=1054.779,63.899,423.021,171.212,31.709,155.936
C02512=1054.773,63.651,423.038,171.210,31.707,155.935
C02513=1054.766,63.401,423.055,171.209,31.704,155.935
C02514=1054.760,63.151,423.073,171.207,31.702,155.934
C02515=1054.753,62.903,423.090,171.206,31.700,155.934
C02516=1054.747,62.653,423.108,171.205,31.698,155.934
C02517=1054.741,62.404,423.125,171.203,31.696,155.933
C02518=1054.734,62.118,423.145,171.201,31.693,155.933
C02519=1054.726,61.833,423.165,171.199,31.690,155.933
C02520=1054.720,61.548,423.185,171.197,31.688,155.932
C02521=1054.713,61.263,423.205,171.195,31.685,155.932
C02522=1054.706,61.013,423.222,171.194,31.683,155.932
C02523=1054.700,60.764,423.239,171.192,31.681,155.931
C02524=1054.694,60.514,423.257,171.191,31.679,155.931
C02525=1054.687,60.266,423.274,171.190,31.677,155.931
C02526=1054.681,60.016,423.292,171.188,31.674,155.930
C02527=1054.675,59.767,423.309,171.186,31.672,155.930
C02528=1054.669,59.517,423.327,171.184,31.669,155.929
C02529=1054.663,59.268,423.343,171.183,31.667,155.929
C02530=1054.656,59.019,423.360,171.181,31.665,155.929
C02531=1054.650,58.770,423.378,171.179,31.663,155.928
C02532=1054.644,58.520,423.395,171.178,31.661,155.928
C02533=1054.638,58.271,423.413,171.177,31.659,155.928
C02534=1054.632,58.021,423.429,171.175,31.656,155.927
C02535=1054.625,57.772,423.446,171.174,31.654,155.927
C02536=1054.619,57.523,423.464,171.172,31.652,155.927
C02537=1054.613,57.274,423.481,171.170,31.649,155.926
C02538=1054.607,57.024,423.499,171.169,31.647,155.926
C02539=1054.601,56.775,423.515,171.167,31.645,155.926
C02540=1054.594,56.525,423.533,171.165,31.643,155.925
C02541=1054.588,56.276,423.550,171.164,31.641,155.925
C02542=1054.582,56.027,423.568,171.163,31.639,155.925
C02543=1054.576,55.777,423.584,171.161,31.636,155.924
C02544=1054.570,55.528,423.601,171.160,31.634,155.924
C02545=1054.563,55.279,423.619,171.158,31.631,155.924
C02546=1054.558,55.029,423.636,171.156,31.629,155.923
C02547=1054.551,54.780,423.653,171.154,31.627,155.923
C02548=1054.545,54.531,423.670,171.153,31.625,155.923
C02549=1054.539,54.281,423.687,171.151,31.622,155.922
C02550=1054.533,54.032,423.704,171.149,31.620,155.922
C02551=1054.527,53.783,423.722,171.149,31.618,155.922
C02552=1054.521,53.533,423.738,171.147,31.616,155.921
C02553=1054.515,53.284,423.755,171.145,31.613,155.921
C02554=1054.508,53.035,423.773,171.144,31.611,155.921
C02555=1054.502,52.785,423.789,171.142,31.609,155.920
C02556=1054.496,52.536,423.806,171.140,31.606,155.920
C02557=1054.490,52.287,423.824,171.139,31.604,155.920
C02558=1054.484,52.037,423.841,171.137,31.602,155.919
C02559=1054.478,51.789,423.858,171.136,31.600,155.919
C02560=1054.472,51.538,423.875,171.135,31.598,155.919
C02561=1054.466,51.290,423.892,171.133,31.595,155.918
C02562=1054.459,51.040,423.909,171.131,31.593,155.918
C02563=1054.454,50.790,423.926,171.130,31.591,155.918
C02564=1054.448,50.542,423.943,171.128,31.588,155.917
C02565=1054.441,50.292,423.960,171.126,31.586,155.917
C02566=1054.435,50.043,423.977,171.125,31.584,155.916
C02567=1054.429,49.793,423.993,171.123,31.582,155.916
C02568=1054.423,49.544,424.011,171.122,31.580,155.916
C02569=1054.417,49.294,424.028,171.121,31.577,155.915
C02570=1054.411,49.045,424.045,171.119,31.575,155.915
C02571=1054.405,48.795,424.061,171.117,31.572,155.915
C02572=1054.399,48.546,424.079,171.116,31.570,155.914
C02573=1054.393,48.297,424.095,171.114,31.568,155.914
C02574=1054.387,48.048,424.112,171.112,31.565,155.914
C02575=1054.381,47.798,424.129,171.111,31.564,155.913
C02576=1054.375,47.549,424.146,171.110,31.561,155.913
C02577=1054.369,47.300,424.162,171.108,31.559,155.913
C02578=1054.363,47.050,424.180,171.106,31.557,155.912
C02579=1054.357,46.801,424.197,171.105,31.554,155.912
C02580=1054.351,46.552,424.214,171.103,31.552,155.912
C02581=1054.345,46.303,424.230,171.101,31.549,155.911
C02582=1054.338,46.017,424.250,171.100,31.547,155.911
C02583=1054.332,45.731,424.269,171.098,31.544,155.910
C02584=1054.324,45.445,424.288,171.096,31.542,155.910
C02585=1054.317,45.160,424.308,171.095,31.539,155.910
C02586=1054.311,44.910,424.324,171.093,31.537,155.909
C02587=1054.305,44.661,424.341,171.091,31.535,155.909
C02588=1054.299,44.412,424.358,171.090,31.532,155.909
C02589=1054.294,44.162,424.374,171.088,31.530,155.908
C02590=1054.287,43.913,424.392,171.086,31.528,155.908
C02591=1054.281,43.664,424.408,171.085,31.525,155.908
C02592=1054.275,43.414,424.424,171.083,31.523,155.907
C02593=1054.269,43.165,424.442,171.082,31.520,155.907
C02594=1054.263,42.915,424.458,171.081,31.519,155.907
C02595=1054.257,42.666,424.475,171.079,31.516,155.906
C02596=1054.250,42.417,424.492,171.077,31.514,155.906
C02597=1054.245,42.168,424.508,171.076,31.512,155.906
C02598=1054.238,41.918,424.524,171.074,31.510,155.905
C02599=1054.232,41.668,424.541,171.072,31.508,155.905
C02600=1054.226,41.420,424.558,171.070,31.505,155.905
C02601=1054.220,41.170,424.574,171.070,31.503,155.904
C02602=1054.213,40.920,424.591,171.068,31.501,155.904
C02603=1054.207,40.671,424.607,171.066,31.498,155.904
C02604=1054.201,40.422,424.624,171.065,31.496,155.903
C02605=1054.195,40.173,424.640,171.063,31.494,155.903
C02606=1054.189,39.923,424.657,171.061,31.492,155.903
C02607=1054.183,39.673,424.673,171.060,31.490,155.902
C02608=1054.177,39.424,424.689,171.058,31.487,155.902
C02609=1054.170,39.175,424.706,171.057,31.485,155.902
C02610=1054.164,38.926,424.722,171.056,31.483,155.901
C02611=1054.158,38.676,424.739,171.054,31.481,155.901
C02612=1054.152,38.426,424.755,171.052,31.479,155.901
C02613=1054.146,38.177,424.772,171.050,31.476,155.900
C02614=1054.141,37.927,424.788,171.049,31.474,155.900
C02615=1054.134,37.679,424.805,171.047,31.472,155.900
C02616=1054.128,37.430,424.821,171.045,31.470,155.899
C02617=1054.121,37.180,424.838,171.045,31.467,155.899
C02618=1054.115,36.930,424.854,171.043,31.465,155.899
C02619=1054.109,36.681,424.870,171.041,31.463,155.898
C02620=1054.103,36.432,424.886,171.040,31.461,155.898
C02621=1054.097,36.182,424.903,171.038,31.459,155.898
C02622=1054.090,35.933,424.919,171.036,31.456,155.897
C02623=1054.084,35.683,424.935,171.034,31.454,155.897
C02624=1054.078,35.434,424.951,171.033,31.452,155.897
C02625=1054.072,35.184,424.967,171.032,31.450,155.896
C02626=1054.066,34.935,424.984,171.030,31.448,155.896
C02627=1054.060,34.685,425.000,171.029,31.445,155.896
C02628=1054.053,34.436,425.016,171.027,31.443,155.895
C02629=1054.047,34.187,425.032,171.025,31.441,155.895
C02630=1054.041,33.937,425.049,171.023,31.439,155.895
C02631=1054.035,33.688,425.065,171.022,31.437,155.894
C02632=1054.029,33.439,425.081,171.020,31.435,155.894
C02633=1054.022,33.189,425.097,171.019,31.432,155.894
C02634=1054.016,32.940,425.113,171.018,31.431,155.894
C02635=1054.010,32.690,425.130,171.016,31.428,155.893
C02636=1054.004,32.441,425.146,171.014,31.426,155.893
C02637=1053.998,32.192,425.162,171.012,31.424,155.893
C02638=1053.992,31.942,425.178,171.011,31.422,155.892
C02639=1053.986,31.693,425.194,171.009,31.420,155.892
C02640=1053.980,31.444,425.210,171.007,31.417,155.892
C02641=1053.974,31.194,425.227,171.007,31.415,155.891
C02642=1053.967,30.944,425.243,171.005,31.413,155.891
C02643=1053.960,30.695,425.259,171.003,31.411,155.891
C02644=1053.955,30.446,425.275,171.001,31.409,155.890
C02645=1053.949,30.197,425.291,171.000,31.406,155.890
C02646=1053.942,29.911,425.310,170.998,31.404,155.890
C02647=1053.935,29.626,425.328,170.996,31.401,155.889
C02648=1053.928,29.339,425.346,170.994,31.399,155.889
C02649=1053.921,29.054,425.365,170.993,31.396,155.889
C02650=1053.915,28.804,425.381,170.991,31.394,155.888
C02651=1053.908,28.555,425.397,170.989,31.392,155.888
C02652=1053.902,28.305,425.412,170.988,31.390,155.888
C02653=1053.897,28.056,425.428,170.986,31.388,155.887
C02654=1053.890,27.807,425.444,170.984,31.385,155.887
C02655=1053.884,27.558,425.460,170.983,31.384,155.887
C02656=1053.877,27.309,425.476,170.982,31.381,155.886
C02657=1053.871,27.058,425.492,170.980,31.379,155.886
C02658=1053.865,26.809,425.508,170.978,31.377,155.886
C02659=1053.858,26.560,425.524,170.977,31.375,155.885
C02660=1053.852,26.310,425.540,170.975,31.373,155.885
C02661=1053.847,26.060,425.556,170.973,31.370,155.885
C02662=1053.840,25.811,425.571,170.971,31.368,155.884
C02663=1053.834,25.562,425.588,170.970,31.366,155.884
C02664=1053.827,25.313,425.603,170.969,31.364,155.884
C02665=1053.822,25.063,425.619,170.967,31.362,155.883
C02666=1053.815,24.814,425.634,170.966,31.360,155.883
C02667=1053.809,24.565,425.651,170.964,31.358,155.883
C02668=1053.803,24.315,425.666,170.962,31.355,155.883
C02669=1053.797,24.066,425.682,170.960,31.353,155.882
C02670=1053.791,23.816,425.698,170.959,31.351,155.882
C02671=1053.784,23.567,425.713,170.957,31.349,155.882
C02672=1053.778,23.317,425.729,170.956,31.347,155.881
C02673=1053.772,23.068,425.745,170.954,31.344,155.881
C02674=1053.766,22.818,425.761,170.953,31.343,155.881
C02675=1053.759,22.569,425.776,170.951,31.340,155.880
C02676=1053.754,22.320,425.793,170.949,31.338,155.880
C02677=1053.747,22.070,425.807,170.947,31.336,155.880
C02678=1053.741,21.821,425.824,170.946,31.334,155.880
C02679=1053.736,21.571,425.839,170.944,31.332,155.879
C02680=1053.729,21.322,425.855,170.943,31.329,155.879
C02681=1053.723,21.072,425.871,170.942,31.327,155.879
C02682=1053.717,20.823,425.886,170.940,31.325,155.878
C02683=1053.711,20.573,425.902,170.938,31.323,155.878
C02684=1053.704,20.324,425.917,170.936,31.321,155.878
C02685=1053.698,20.074,425.934,170.935,31.319,155.877
C02686=1053.692,19.825,425.949,170.933,31.317,155.877
C02687=1053.686,19.575,425.965,170.931,31.315,155.877
C02688=1053.679,19.326,425.980,170.930,31.313,155.876
C02689=1053.673,19.077,425.995,170.929,31.311,155.876
C02690=1053.667,18.827,426.012,170.927,31.309,155.876
C02691=1053.660,18.578,426.027,170.925,31.307,155.876
C02692=1053.655,18.328,426.043,170.923,31.304,155.875
C02693=1053.648,18.079,426.058,170.922,31.302,155.875
C02694=1053.641,17.830,426.073,170.920,31.300,155.875
C02695=1053.636,17.580,426.089,170.919,31.298,155.874
C02696=1053.630,17.331,426.104,170.917,31.296,155.874
C02697=1053.624,17.081,426.120,170.916,31.294,155.874
C02698=1053.618,16.832,426.135,170.914,31.292,155.873
C02699=1053.611,16.583,426.150,170.912,31.290,155.873
C02700=1053.605,16.333,426.166,170.910,31.287,155.873
C02701=1053.599,16.084,426.182,170.909,31.285,155.873
C02702=1053.593,15.834,426.197,170.907,31.283,155.872
C02703=1053.587,15.584,426.212,170.906,31.281,155.872
C02704=1053.580,15.335,426.228,170.904,31.279,155.872
C02705=1053.574,15.085,426.243,170.903,31.277,155.871
C02706=1053.568,14.837,426.259,170.901,31.275,155.871
C02707=1053.562,14.587,426.274,170.899,31.273,155.871
C02708=1053.556,14.337,426.289,170.897,31.271,155.871
C02709=1053.550,14.088,426.305,170.895,31.269,155.870
C02710=1053.542,13.781,426.323,170.894,31.266,155.870
C02711=1053.534,13.475,426.342,170.892,31.263,155.869
C02712=1053.526,13.170,426.361,170.890,31.261,155.869
C02713=1053.518,12.863,426.379,170.888,31.258,155.869
C02714=1053.512,12.624,426.394,170.886,31.256,155.868
C02715=1053.507,12.386,426.408,170.884,31.255,155.868
C02716=1053.501,12.147,426.423,170.883,31.253,155.868
C02717=1053.494,11.909,426.438,170.882,31.251,155.868
C02718=1053.489,11.671,426.452,170.880,31.249,155.867
C02719=1053.482,11.432,426.467,170.879,31.247,155.867
C02720=1053.476,11.193,426.481,170.877,31.245,155.867
C02721=1053.470,10.955,426.496,170.875,31.243,155.867
C02722=1053.464,10.705,426.511,170.873,31.241,155.866
C02723=1053.458,10.456,426.526,170.872,31.239,155.866
C02724=1053.452,10.206,426.541,170.870,31.237,155.866
C02725=1053.445,9.957,426.556,170.869,31.235,155.865
C02726=1053.439,9.707,426.571,170.867,31.233,155.865
C02727=1053.433,9.458,426.586,170.865,31.231,155.865
C02728=1053.426,9.208,426.601,170.864,31.229,155.865
C02729=1053.420,8.959,426.616,170.862,31.226,155.864
C02730=1053.415,8.709,426.631,170.860,31.225,155.864
C02731=1053.408,8.460,426.647,170.858,31.223,155.864
C02732=1053.402,8.210,426.662,170.857,31.221,155.864
C02733=1053.395,7.961,426.677,170.856,31.219,155.863
C02734=1053.389,7.711,426.692,170.854,31.217,155.863
C02735=1053.383,7.462,426.707,170.852,31.215,155.863
C02736=1053.377,7.213,426.721,170.850,31.212,155.862
C02737=1053.370,6.963,426.736,170.849,31.210,155.862
C02738=1053.364,6.714,426.752,170.847,31.208,155.862
C02739=1053.358,6.464,426.768,170.845,31.206,155.862
C02740=1053.352,6.215,426.782,170.844,31.204,155.861
C02741=1053.346,5.965,426.797,170.842,31.202,155.861
C02742=1053.339,5.716,426.812,170.841,31.200,155.861
C02743=1053.333,5.466,426.827,170.839,31.198,155.860
C02744=1053.327,5.217,426.842,170.837,31.196,155.860
C02745=1053.321,4.967,426.857,170.835,31.194,155.860
C02746=1053.314,4.718,426.871,170.834,31.192,155.860
C02747=1053.308,4.468,426.886,170.833,31.190,155.859
C02748=1053.302,4.219,426.901,170.831,31.188,155.859
C02749=1053.296,3.969,426.916,170.829,31.186,155.859
C02750=1053.290,3.719,426.932,170.827,31.184,155.858
C02751=1053.284,3.470,426.946,170.826,31.182,155.858
C02752=1053.278,3.221,426.961,170.824,31.180,155.858
C02753=1053.272,2.971,426.976,170.822,31.178,155.858
C02754=1053.265,2.722,426.991,170.820,31.176,155.857
C02755=1053.260,2.473,427.006,170.819,31.174,155.857
C02756=1053.253,2.223,427.020,170.818,31.172,155.857
C02757=1053.247,1.973,427.035,170.816,31.170,155.857
C02758=1053.240,1.724,427.050,170.814,31.168,155.856
C02759=1053.235,1.475,427.065,170.812,31.166,155.856
C02760=1053.228,1.225,427.080,170.810,31.164,155.856
C02761=1053.222,0.975,427.095,170.809,31.162,155.855
C02762=1053.216,0.726,427.109,170.808,31.159,155.855
C02763=1053.210,0.477,427.124,170.806,31.157,155.855
C02764=1053.203,0.227,427.139,170.804,31.155,155.854
C02765=1053.198,-0.022,427.154,170.802,31.153,155.854
C02766=1053.191,-0.272,427.168,170.801,31.152,155.854
C02767=1053.185,-0.522,427.183,170.799,31.150,155.854
C02768=1053.180,-0.771,427.198,170.797,31.147,155.853
C02769=1053.174,-1.021,427.213,170.796,31.145,155.853
C02770=1053.168,-1.270,427.228,170.794,31.143,155.853
C02771=1053.162,-1.519,427.243,170.793,31.141,155.853
C02772=1053.155,-1.769,427.258,170.791,31.139,155.852
C02773=1053.149,-2.018,427.272,170.789,31.137,155.852
C02774=1053.142,-2.301,427.289,170.787,31.135,155.852
C02775=1053.135,-2.584,427.305,170.785,31.133,155.851
C02776=1053.129,-2.866,427.322,170.784,31.130,155.851
C02777=1053.122,-3.148,427.339,170.782,31.128,155.851
C02778=1053.116,-3.398,427.353,170.780,31.126,155.850
C02779=1053.109,-3.648,427.367,170.778,31.124,155.850
C02780=1053.103,-3.896,427.382,170.776,31.122,155.850
C02781=1053.097,-4.146,427.397,170.774,31.120,155.850
C02782=1053.090,-4.396,427.411,170.773,31.118,155.849
C02783=1053.084,-4.645,427.425,170.772,31.117,155.849
C02784=1053.078,-4.895,427.440,170.770,31.114,155.849
C02785=1053.071,-5.144,427.455,170.768,31.112,155.849
C02786=1053.066,-5.394,427.469,170.766,31.110,155.848
C02787=1053.059,-5.643,427.483,170.764,31.109,155.848
C02788=1053.052,-5.893,427.498,170.763,31.107,155.848
C02789=1053.047,-6.143,427.512,170.761,31.105,155.848
C02790=1053.040,-6.392,427.526,170.759,31.103,155.847
C02791=1053.034,-6.641,427.541,170.758,31.101,155.847
C02792=1053.028,-6.891,427.555,170.756,31.099,155.847
C02793=1053.021,-7.141,427.570,170.754,31.097,155.847
C02794=1053.015,-7.389,427.584,170.752,31.095,155.846
C02795=1053.009,-7.640,427.598,170.751,31.093,155.846
C02796=1053.003,-7.889,427.613,170.749,31.091,155.846
C02797=1052.996,-8.139,427.626,170.747,31.090,155.846
C02798=1052.990,-8.388,427.641,170.746,31.087,155.845
C02799=1052.984,-8.637,427.656,170.744,31.085,155.845
C02800=1052.978,-8.887,427.670,170.742,31.083,155.845
C02801=1052.971,-9.136,427.684,170.741,31.082,155.845
C02802=1052.965,-9.386,427.698,170.739,31.080,155.844
C02803=1052.960,-9.635,427.713,170.737,31.078,155.844
C02804=1052.952,-9.885,427.727,170.735,31.076,155.844
C02805=1052.947,-10.134,427.741,170.734,31.074,155.844
C02806=1052.941,-10.384,427.756,170.732,31.072,155.843
C02807=1052.934,-10.634,427.770,170.730,31.070,155.843
C02808=1052.928,-10.883,427.784,170.729,31.068,155.843
C02809=1052.922,-11.133,427.799,170.727,31.066,155.843
C02810=1052.915,-11.382,427.813,170.725,31.064,155.842
C02811=1052.909,-11.632,427.827,170.723,31.063,155.842
C02812=1052.904,-11.881,427.841,170.722,31.060,155.842
C02813=1052.897,-12.131,427.856,170.720,31.058,155.842
C02814=1052.891,-12.380,427.870,170.718,31.057,155.841
C02815=1052.885,-12.630,427.884,170.717,31.055,155.841
C02816=1052.879,-12.879,427.898,170.715,31.053,155.841
C02817=1052.872,-13.129,427.912,170.713,31.051,155.841
C02818=1052.866,-13.378,427.927,170.711,31.049,155.840
C02819=1052.860,-13.628,427.941,170.710,31.047,155.840
C02820=1052.854,-13.878,427.954,170.708,31.045,155.840
C02821=1052.848,-14.127,427.969,170.706,31.043,155.840
C02822=1052.842,-14.377,427.982,170.705,31.041,155.839
C02823=1052.836,-14.625,427.997,170.703,31.040,155.839
C02824=1052.830,-14.876,428.011,170.701,31.038,155.839
C02825=1052.823,-15.124,428.025,170.699,31.035,155.839
C02826=1052.817,-15.375,428.039,170.697,31.034,155.838
C02827=1052.811,-15.624,428.053,170.696,31.032,155.838
C02828=1052.805,-15.874,428.068,170.694,31.030,155.838
C02829=1052.798,-16.123,428.081,170.692,31.028,155.838
C02830=1052.792,-16.373,428.095,170.691,31.026,155.837
C02831=1052.786,-16.622,428.109,170.689,31.025,155.837
C02832=1052.780,-16.872,428.123,170.687,31.022,155.837
C02833=1052.773,-17.121,428.137,170.685,31.021,155.837
C02834=1052.766,-17.371,428.151,170.684,31.019,155.837
C02835=1052.761,-17.620,428.165,170.682,31.017,155.836
C02836=1052.754,-17.870,428.178,170.680,31.015,155.836
C02837=1052.749,-18.120,428.192,170.678,31.014,155.836
C02838=1052.741,-18.400,428.208,170.676,31.012,155.836
C02839=1052.734,-18.681,428.224,170.674,31.009,155.835
C02840=1052.727,-18.962,428.240,170.672,31.007,155.835
C02841=1052.720,-19.243,428.255,170.671,31.005,155.835
C02842=1052.714,-19.493,428.269,170.669,31.004,155.835
C02843=1052.708,-19.742,428.283,170.667,31.001,155.834
C02844=1052.701,-19.991,428.297,170.665,31.000,155.834
C02845=1052.695,-20.241,428.310,170.663,30.998,155.834
C02846=1052.689,-20.490,428.324,170.661,30.996,155.834
C02847=1052.682,-20.740,428.338,170.659,30.994,155.833
C02848=1052.677,-20.990,428.352,170.659,30.993,155.833
C02849=1052.670,-21.239,428.366,170.657,30.991,155.833
C02850=1052.664,-21.488,428.379,170.655,30.989,155.833
C02851=1052.658,-21.738,428.393,170.653,30.987,155.833
C02852=1052.651,-21.988,428.407,170.651,30.985,155.832
C02853=1052.646,-22.238,428.420,170.649,30.983,155.832
C02854=1052.640,-22.487,428.434,170.647,30.982,155.832
C02855=1052.633,-22.737,428.447,170.646,30.980,155.832
C02856=1052.627,-22.986,428.462,170.644,30.978,155.831
C02857=1052.620,-23.236,428.476,170.642,30.976,155.831
C02858=1052.614,-23.485,428.489,170.641,30.975,155.831
C02859=1052.609,-23.735,428.503,170.639,30.972,155.831
C02860=1052.602,-23.985,428.516,170.637,30.971,155.831
C02861=1052.596,-24.234,428.530,170.635,30.969,155.830
C02862=1052.590,-24.483,428.544,170.634,30.967,155.830
C02863=1052.583,-24.733,428.557,170.632,30.965,155.830
C02864=1052.578,-24.983,428.571,170.630,30.964,155.830
C02865=1052.572,-25.232,428.584,170.628,30.961,155.829
C02866=1052.565,-25.481,428.598,170.626,30.960,155.829
C02867=1052.559,-25.732,428.612,170.624,30.958,155.829
C02868=1052.553,-25.980,428.626,170.622,30.956,155.829
C02869=1052.547,-26.230,428.639,170.622,30.954,155.828
C02870=1052.540,-26.480,428.653,170.620,30.953,155.828
C02871=1052.534,-26.729,428.667,170.618,30.951,155.828
C02872=1052.528,-26.978,428.680,170.616,30.949,155.828
C02873=1052.522,-27.229,428.693,170.614,30.948,155.828
C02874=1052.516,-27.479,428.707,170.612,30.945,155.827
C02875=1052.510,-27.728,428.720,170.610,30.944,155.827
C02876=1052.503,-27.978,428.733,170.608,30.942,155.827
C02877=1052.497,-28.227,428.747,170.607,30.940,155.827
C02878=1052.491,-28.476,428.760,170.605,30.939,155.827
C02879=1052.484,-28.726,428.773,170.603,30.937,155.826
C02880=1052.478,-28.976,428.787,170.601,30.935,155.826
C02881=1052.472,-29.225,428.801,170.599,30.934,155.826
C02882=1052.466,-29.474,428.814,170.597,30.932,155.826
C02883=1052.459,-29.724,428.828,170.595,30.930,155.826
C02884=1052.453,-29.974,428.841,170.595,30.928,155.825
C02885=1052.447,-30.223,428.854,170.593,30.927,155.825
C02886=1052.441,-30.473,428.867,170.591,30.925,155.825
C02887=1052.434,-30.723,428.880,170.589,30.923,155.825
C02888=1052.428,-30.972,428.894,170.587,30.922,155.825
C02889=1052.421,-31.221,428.907,170.585,30.920,155.824
C02890=1052.416,-31.471,428.921,170.583,30.918,155.824
C02891=1052.409,-31.721,428.934,170.582,30.917,155.824
C02892=1052.403,-31.971,428.947,170.580,30.915,155.824
C02893=1052.397,-32.220,428.960,170.578,30.913,155.824
C02894=1052.391,-32.469,428.974,170.576,30.911,155.823
C02895=1052.384,-32.719,428.987,170.574,30.910,155.823
C02896=1052.378,-32.968,429.000,170.572,30.908,155.823
C02897=1052.372,-33.218,429.013,170.570,30.906,155.823
C02898=1052.366,-33.468,429.026,170.568,30.905,155.823
C02899=1052.359,-33.717,429.040,170.567,30.903,155.822
C02900=1052.353,-33.967,429.053,170.565,30.901,155.822
C02901=1052.347,-34.217,429.066,170.563,30.899,155.822
C02902=1052.340,-34.497,429.081,170.561,30.897,155.822
C02903=1052.333,-34.777,429.096,170.559,30.896,155.822
C02904=1052.326,-35.057,429.111,170.557,30.894,155.821
C02905=1052.319,-35.337,429.125,170.555,30.892,155.821
C02906=1052.313,-35.587,429.139,170.554,30.890,155.821
C02907=1052.307,-35.836,429.152,170.552,30.888,155.821
C02908=1052.301,-36.086,429.165,170.550,30.887,155.821
C02909=1052.295,-36.335,429.178,170.548,30.885,155.820
C02910=1052.288,-36.584,429.191,170.546,30.883,155.820
C02911=1052.283,-36.834,429.204,170.544,30.882,155.820
C02912=1052.276,-37.084,429.217,170.542,30.880,155.820
C02913=1052.270,-37.333,429.231,170.541,30.879,155.820
C02914=1052.264,-37.583,429.243,170.539,30.876,155.819
C02915=1052.258,-37.833,429.257,170.537,30.875,155.819
C02916=1052.252,-38.082,429.270,170.535,30.873,155.819
C02917=1052.246,-38.332,429.283,170.533,30.872,155.819
C02918=1052.240,-38.581,429.296,170.531,30.870,155.819
C02919=1052.234,-38.831,429.309,170.529,30.868,155.818
C02920=1052.226,-39.081,429.322,170.528,30.867,155.818
C02921=1052.220,-39.330,429.335,170.526,30.865,155.818
C02922=1052.214,-39.580,429.347,170.524,30.863,155.818
C02923=1052.208,-39.829,429.361,170.522,30.862,155.818
C02924=1052.202,-40.079,429.373,170.520,30.860,155.818
C02925=1052.196,-40.328,429.387,170.518,30.859,155.817
C02926=1052.189,-40.578,429.399,170.516,30.857,155.817
C02927=1052.183,-40.827,429.412,170.515,30.856,155.817
C02928=1052.176,-41.078,429.425,170.513,30.854,155.817
C02929=1052.170,-41.327,429.438,170.511,30.852,155.817
C02930=1052.164,-41.577,429.451,170.509,30.851,155.816
C02931=1052.157,-41.826,429.463,170.507,30.849,155.816
C02932=1052.152,-42.076,429.476,170.505,30.848,155.816
C02933=1052.145,-42.325,429.489,170.503,30.846,155.816
C02934=1052.139,-42.575,429.502,170.501,30.844,155.816
C02935=1052.133,-42.824,429.515,170.500,30.843,155.816
C02936=1052.127,-43.074,429.527,170.498,30.841,155.815
C02937=1052.120,-43.323,429.540,170.496,30.840,155.815
C02938=1052.114,-43.573,429.553,170.494,30.838,155.815
C02939=1052.108,-43.823,429.565,170.492,30.837,155.815
C02940=1052.102,-44.072,429.578,170.490,30.835,155.815
C02941=1052.095,-44.322,429.591,170.488,30.834,155.815
C02942=1052.089,-44.572,429.604,170.487,30.832,155.815
C02943=1052.083,-44.821,429.617,170.485,30.830,155.814
C02944=1052.077,-45.071,429.629,170.483,30.828,155.814
C02945=1052.071,-45.321,429.642,170.481,30.827,155.814
C02946=1052.064,-45.570,429.654,170.479,30.825,155.814
C02947=1052.058,-45.819,429.668,170.477,30.824,155.814
C02948=1052.052,-46.069,429.680,170.475,30.822,155.813
C02949=1052.046,-46.319,429.693,170.473,30.821,155.813
C02950=1052.040,-46.568,429.706,170.472,30.819,155.813
C02951=1052.033,-46.818,429.718,170.470,30.818,155.813
C02952=1052.027,-47.068,429.731,170.468,30.816,155.813
C02953=1052.021,-47.317,429.744,170.466,30.815,155.813
C02954=1052.015,-47.567,429.756,170.464,30.813,155.812
C02955=1052.009,-47.817,429.768,170.462,30.812,155.812
C02956=1052.003,-48.067,429.781,170.460,30.810,155.812
C02957=1051.996,-48.316,429.794,170.459,30.808,155.812
C02958=1051.991,-48.565,429.806,170.457,30.807,155.812
C02959=1051.984,-48.815,429.818,170.455,30.805,155.812
C02960=1051.979,-49.064,429.831,170.453,30.804,155.811
C02961=1051.972,-49.314,429.844,170.451,30.802,155.811
C02962=1051.966,-49.564,429.857,170.449,30.801,155.811
C02963=1051.960,-49.813,429.869,170.447,30.799,155.811
C02964=1051.954,-50.063,429.881,170.445,30.798,155.811
C02965=1051.948,-50.312,429.894,170.444,30.796,155.811
C02966=1051.940,-50.593,429.908,170.442,30.795,155.810
C02967=1051.933,-50.873,429.922,170.440,30.793,155.810
C02968=1051.926,-51.154,429.935,170.437,30.791,155.810
C02969=1051.919,-51.435,429.950,170.435,30.790,155.810
C02970=1051.913,-51.684,429.961,170.433,30.788,155.810
C02971=1051.907,-51.934,429.974,170.431,30.787,155.810
C02972=1051.900,-52.184,429.986,170.430,30.786,155.810
C02973=1051.894,-52.433,429.999,170.428,30.784,155.810
C02974=1051.887,-52.682,430.011,170.426,30.783,155.809
C02975=1051.880,-52.932,430.023,170.424,30.782,155.809
C02976=1051.875,-53.182,430.036,170.422,30.780,155.809
C02977=1051.868,-53.431,430.048,170.420,30.779,155.809
C02978=1051.862,-53.681,430.060,170.418,30.777,155.809
C02979=1051.855,-53.931,430.072,170.416,30.776,155.809
C02980=1051.849,-54.181,430.085,170.414,30.774,155.809
C02981=1051.843,-54.430,430.097,170.412,30.773,155.808
C02982=1051.836,-54.680,430.109,170.410,30.771,155.808
C02983=1051.831,-54.929,430.121,170.408,30.770,155.808
C02984=1051.824,-55.179,430.133,170.406,30.769,155.808
C02985=1051.818,-55.429,430.145,170.404,30.767,155.808
C02986=1051.812,-55.678,430.157,170.402,30.766,155.808
C02987=1051.805,-55.928,430.169,170.400,30.765,155.808
C02988=1051.799,-56.178,430.182,170.399,30.763,155.808
C02989=1051.792,-56.427,430.194,170.397,30.762,155.807
C02990=1051.786,-56.677,430.206,170.395,30.761,155.807
C02991=1051.780,-56.927,430.218,170.393,30.759,155.807
C02992=1051.773,-57.176,430.230,170.391,30.758,155.807
C02993=1051.768,-57.425,430.242,170.389,30.756,155.807
C02994=1051.761,-57.675,430.254,170.387,30.755,155.807
C02995=1051.755,-57.924,430.266,170.385,30.754,155.807
C02996=1051.749,-58.174,430.279,170.384,30.752,155.806
C02997=1051.742,-58.424,430.291,170.381,30.751,155.806
C02998=1051.735,-58.673,430.303,170.379,30.750,155.806
C02999=1051.730,-58.923,430.315,170.377,30.748,155.806
C03000=1051.724,-59.172,430.327,170.375,30.747,155.806
C03001=1051.718,-59.423,430.339,170.373,30.746,155.806
C03002=1051.711,-59.672,430.351,170.371,30.744,155.806
C03003=1051.705,-59.922,430.363,170.369,30.743,155.806
C03004=1051.699,-60.172,430.375,170.368,30.742,155.806
C03005=1051.693,-60.421,430.387,170.366,30.740,155.805
C03006=1051.686,-60.670,430.399,170.364,30.739,155.805
C03007=1051.680,-60.920,430.411,170.362,30.738,155.805
C03008=1051.674,-61.170,430.423,170.360,30.736,155.805
C03009=1051.667,-61.420,430.435,170.358,30.735,155.805
C03010=1051.662,-61.669,430.447,170.356,30.733,155.805
C03011=1051.655,-61.919,430.459,170.354,30.732,155.805
C03012=1051.649,-62.168,430.471,170.352,30.731,155.805
C03013=1051.643,-62.418,430.483,170.350,30.729,155.804
C03014=1051.637,-62.668,430.494,170.348,30.728,155.804
C03015=1051.630,-62.917,430.506,170.346,30.727,155.804
C03016=1051.624,-63.167,430.519,170.344,30.725,155.804
C03017=1051.618,-63.417,430.531,170.342,30.724,155.804
C03018=1051.612,-63.666,430.542,170.340,30.723,155.804
C03019=1051.606,-63.916,430.554,170.339,30.721,155.804
C03020=1051.599,-64.166,430.566,170.337,30.720,155.804
C03021=1051.593,-64.415,430.578,170.335,30.719,155.804
C03022=1051.587,-64.665,430.589,170.333,30.718,155.803
C03023=1051.581,-64.914,430.601,170.331,30.716,155.803
C03024=1051.574,-65.164,430.613,170.329,30.715,155.803
C03025=1051.569,-65.414,430.624,170.326,30.714,155.803
C03026=1051.563,-65.663,430.637,170.324,30.712,155.803
C03027=1051.556,-65.913,430.649,170.322,30.711,155.803
C03028=1051.550,-66.162,430.660,170.321,30.710,155.803
C03029=1051.544,-66.412,430.672,170.319,30.709,155.803
C03030=1051.537,-66.694,430.685,170.317,30.707,155.803
C03031=1051.530,-66.975,430.699,170.314,30.705,155.802
C03032=1051.523,-67.257,430.712,170.312,30.704,155.802
C03033=1051.516,-67.540,430.725,170.310,30.702,155.802
C03034=1051.510,-67.789,430.737,170.308,30.701,155.802
C03035=1051.504,-68.039,430.749,170.307,30.700,155.802
C03036=1051.498,-68.288,430.760,170.305,30.699,155.802
C03037=1051.492,-68.538,430.772,170.302,30.697,155.802
C03038=1051.486,-68.788,430.784,170.300,30.696,155.802
C03039=1051.480,-69.037,430.795,170.298,30.695,155.802
C03040=1051.473,-69.287,430.806,170.296,30.694,155.801
C03041=1051.467,-69.537,430.819,170.294,30.692,155.801
C03042=1051.461,-69.786,430.831,170.292,30.691,155.801
C03043=1051.455,-70.036,430.842,170.291,30.690,155.801
C03044=1051.449,-70.285,430.853,170.289,30.689,155.801
C03045=1051.443,-70.536,430.865,170.287,30.687,155.801
C03046=1051.437,-70.785,430.877,170.285,30.686,155.801
C03047=1051.431,-71.035,430.888,170.283,30.685,155.801
C03048=1051.424,-71.284,430.900,170.280,30.684,155.801
C03049=1051.419,-71.534,430.912,170.278,30.682,155.801
C03050=1051.413,-71.784,430.924,170.276,30.681,155.800
C03051=1051.407,-72.033,430.934,170.275,30.680,155.800
C03052=1051.400,-72.283,430.946,170.273,30.679,155.800
C03053=1051.395,-72.533,430.958,170.271,30.677,155.800
C03054=1051.389,-72.782,430.970,170.269,30.676,155.800
C03055=1051.382,-73.032,430.981,170.267,30.675,155.800
C03056=1051.376,-73.281,430.993,170.265,30.674,155.800
C03057=1051.370,-73.531,431.004,170.263,30.672,155.800
C03058=1051.365,-73.781,431.015,170.260,30.671,155.800
C03059=1051.358,-74.031,431.027,170.259,30.669,155.800
C03060=1051.353,-74.280,431.038,170.257,30.669,155.799
C03061=1051.346,-74.530,431.050,170.255,30.668,155.799
C03062=1051.340,-74.780,431.061,170.253,30.666,155.799
C03063=1051.334,-75.029,431.072,170.251,30.665,155.799
C03064=1051.327,-75.279,431.084,170.249,30.664,155.799
C03065=1051.322,-75.528,431.095,170.247,30.663,155.799
C03066=1051.315,-75.779,431.106,170.244,30.662,155.799
C03067=1051.309,-76.027,431.118,170.242,30.661,155.799
C03068=1051.303,-76.278,431.129,170.241,30.660,155.799
C03069=1051.297,-76.527,431.140,170.239,30.658,155.799
C03070=1051.290,-76.777,431.152,170.237,30.657,155.799
C03071=1051.284,-77.027,431.163,170.235,30.656,155.799
C03072=1051.278,-77.276,431.174,170.233,30.655,155.799
C03073=1051.272,-77.526,431.186,170.231,30.654,155.798
C03074=1051.266,-77.775,431.197,170.229,30.653,155.798
C03075=1051.260,-78.026,431.208,170.226,30.652,155.798
C03076=1051.253,-78.275,431.218,170.224,30.651,155.798
C03077=1051.246,-78.524,431.230,170.223,30.649,155.798
C03078=1051.241,-78.774,431.241,170.221,30.648,155.798
C03079=1051.234,-79.024,431.253,170.219,30.647,155.798
C03080=1051.229,-79.274,431.263,170.217,30.646,155.798
C03081=1051.222,-79.523,431.275,170.215,30.645,155.798
C03082=1051.216,-79.773,431.286,170.212,30.644,155.798
C03083=1051.210,-80.023,431.298,170.210,30.643,155.798
C03084=1051.204,-80.272,431.308,170.208,30.642,155.798
C03085=1051.197,-80.522,431.319,170.206,30.641,155.798
C03086=1051.191,-80.772,431.330,170.205,30.640,155.798
C03087=1051.185,-81.021,431.342,170.203,30.639,155.798
C03088=1051.179,-81.271,431.353,170.201,30.638,155.798
C03089=1051.172,-81.521,431.363,170.198,30.637,155.798
C03090=1051.166,-81.770,431.374,170.196,30.636,155.798
C03091=1051.160,-82.020,431.386,170.194,30.635,155.797
C03092=1051.154,-82.270,431.396,170.192,30.634,155.797
C03093=1051.147,-82.520,431.407,170.190,30.633,155.797
C03094=1051.140,-82.804,431.420,170.188,30.632,155.797
C03095=1051.134,-83.087,431.432,170.186,30.631,155.797
C03096=1051.126,-83.371,431.445,170.183,30.629,155.797
C03097=1051.119,-83.655,431.457,170.181,30.629,155.797
C03098=1051.112,-83.905,431.468,170.179,30.628,155.797
C03099=1051.107,-84.154,431.479,170.177,30.627,155.797
C03100=1051.100,-84.405,431.490,170.175,30.626,155.797
C03101=1051.094,-84.654,431.500,170.172,30.625,155.797
C03102=1051.087,-84.904,431.512,170.170,30.624,155.797
C03103=1051.082,-85.153,431.522,170.168,30.623,155.797
C03104=1051.075,-85.403,431.533,170.167,30.622,155.797
C03105=1051.069,-85.653,431.544,170.165,30.621,155.797
C03106=1051.063,-85.902,431.555,170.163,30.620,155.797
C03107=1051.056,-86.152,431.566,170.160,30.619,155.797
C03108=1051.050,-86.402,431.576,170.158,30.618,155.797
C03109=1051.045,-86.651,431.587,170.156,30.617,155.797
C03110=1051.038,-86.901,431.598,170.154,30.616,155.797
C03111=1051.032,-87.151,431.609,170.152,30.615,155.797
C03112=1051.025,-87.401,431.620,170.150,30.614,155.797
C03113=1051.019,-87.650,431.630,170.149,30.613,155.796
C03114=1051.013,-87.899,431.641,170.146,30.612,155.796
C03115=1051.007,-88.150,431.652,170.144,30.611,155.796
C03116=1051.000,-88.399,431.663,170.142,30.610,155.796
C03117=1050.995,-88.649,431.673,170.140,30.609,155.796
C03118=1050.989,-88.899,431.684,170.138,30.609,155.796
C03119=1050.982,-89.148,431.694,170.136,30.608,155.796
C03120=1050.976,-89.398,431.705,170.133,30.607,155.796
C03121=1050.970,-89.648,431.717,170.131,30.606,155.796
C03122=1050.964,-89.897,431.727,170.129,30.605,155.796
C03123=1050.958,-90.147,431.738,170.128,30.604,155.796
C03124=1050.952,-90.397,431.749,170.126,30.603,155.796
C03125=1050.945,-90.647,431.758,170.124,30.602,155.796
C03126=1050.940,-90.896,431.769,170.121,30.601,155.796
C03127=1050.933,-91.146,431.781,170.119,30.600,155.796
C03128=1050.927,-91.395,431.791,170.117,30.600,155.796
C03129=1050.921,-91.645,431.802,170.115,30.599,155.796
C03130=1050.915,-91.895,431.811,170.113,30.598,155.796
C03131=1050.909,-92.145,431.823,170.111,30.597,155.796
C03132=1050.903,-92.394,431.833,170.109,30.596,155.796
C03133=1050.896,-92.644,431.844,170.107,30.595,155.796
C03134=1050.891,-92.893,431.855,170.105,30.594,155.796
C03135=1050.885,-93.144,431.865,170.103,30.594,155.796
C03136=1050.878,-93.393,431.875,170.101,30.593,155.796
C03137=1050.872,-93.643,431.886,170.099,30.592,155.796
C03138=1050.866,-93.892,431.897,170.096,30.591,155.796
C03139=1050.860,-94.143,431.907,170.094,30.590,155.796
C03140=1050.854,-94.392,431.918,170.092,30.589,155.796
C03141=1050.848,-94.641,431.928,170.090,30.588,155.796
C03142=1050.842,-94.891,431.938,170.089,30.587,155.796
C03143=1050.835,-95.141,431.949,170.087,30.587,155.796
C03144=1050.829,-95.391,431.960,170.084,30.585,155.796
C03145=1050.824,-95.640,431.971,170.082,30.584,155.796
C03146=1050.817,-95.890,431.980,170.080,30.584,155.796
C03147=1050.812,-96.139,431.991,170.078,30.583,155.796
C03148=1050.805,-96.389,432.002,170.076,30.582,155.796
C03149=1050.799,-96.639,432.012,170.073,30.581,155.796
C03150=1050.793,-96.889,432.023,170.071,30.580,155.796
C03151=1050.787,-97.139,432.033,170.069,30.580,155.796
C03152=1050.782,-97.388,432.043,170.068,30.579,155.796
C03153=1050.774,-97.638,432.054,170.066,30.578,155.796
C03154=1050.768,-97.888,432.064,170.064,30.578,155.796
C03155=1050.763,-98.137,432.075,170.061,30.577,155.796
C03156=1050.756,-98.387,432.084,170.059,30.576,155.796
C03157=1050.751,-98.637,432.095,170.057,30.575,155.796
C03158=1050.743,-98.923,432.107,170.054,30.574,155.796
C03159=1050.736,-99.209,432.119,170.052,30.573,155.796
C03160=1050.729,-99.495,432.130,170.049,30.573,155.796
C03161=1050.721,-99.782,432.142,170.047,30.572,155.796
C03162=1050.715,-100.032,432.152,170.046,30.571,155.796
C03163=1050.709,-100.281,432.162,170.043,30.570,155.796
C03164=1050.703,-100.531,432.172,170.041,30.569,155.796
C03165=1050.697,-100.780,432.182,170.039,30.569,155.796
C03166=1050.691,-101.030,432.192,170.037,30.568,155.796
C03167=1050.684,-101.280,432.203,170.035,30.568,155.796
C03168=1050.678,-101.530,432.213,170.033,30.567,155.796
C03169=1050.672,-101.780,432.224,170.030,30.566,155.796
C03170=1050.666,-102.029,432.233,170.028,30.565,155.796
C03171=1050.660,-102.279,432.243,170.026,30.565,155.796
C03172=1050.654,-102.529,432.254,170.024,30.564,155.796
C03173=1050.648,-102.778,432.263,170.023,30.563,155.796
C03174=1050.641,-103.028,432.274,170.020,30.563,155.796
C03175=1050.636,-103.278,432.284,170.018,30.562,155.796
C03176=1050.629,-103.528,432.294,170.016,30.562,155.796
C03177=1050.623,-103.777,432.304,170.014,30.561,155.796
C03178=1050.618,-104.028,432.314,170.011,30.560,155.796
C03179=1050.611,-104.277,432.324,170.009,30.559,155.796
C03180=1050.605,-104.527,432.334,170.007,30.559,155.796
C03181=1050.598,-104.776,432.344,170.005,30.558,155.796
C03182=1050.593,-105.026,432.354,170.003,30.558,155.796
C03183=1050.587,-105.276,432.364,170.000,30.557,155.796
C03184=1050.580,-105.525,432.374,169.998,30.556,155.796
C03185=1050.574,-105.776,432.385,169.997,30.556,155.796
C03186=1050.568,-106.025,432.394,169.995,30.555,155.796
C03187=1050.562,-106.275,432.405,169.993,30.555,155.796
C03188=1050.556,-106.524,432.414,169.990,30.553,155.796
C03189=1050.549,-106.774,432.424,169.988,30.553,155.796
C03190=1050.544,-107.024,432.434,169.986,30.553,155.796
C03191=1050.537,-107.273,432.444,169.984,30.552,155.796
C03192=1050.531,-107.523,432.454,169.982,30.551,155.796
C03193=1050.525,-107.773,432.463,169.979,30.551,155.796
C03194=1050.519,-108.023,432.473,169.977,30.550,155.796
C03195=1050.513,-108.272,432.484,169.975,30.550,155.796
C03196=1050.507,-108.522,432.493,169.973,30.549,155.796
C03197=1050.501,-108.772,432.503,169.972,30.548,155.796
C03198=1050.495,-109.022,432.512,169.969,30.548,155.796
C03199=1050.488,-109.271,432.523,169.967,30.548,155.797
C03200=1050.482,-109.521,432.532,169.965,30.547,155.797
C03201=1050.476,-109.771,432.542,169.963,30.546,155.797
C03202=1050.470,-110.020,432.551,169.960,30.546,155.797
C03203=1050.463,-110.270,432.561,169.958,30.546,155.797
C03204=1050.458,-110.520,432.572,169.956,30.545,155.797
C03205=1050.452,-110.769,432.581,169.954,30.544,155.797
C03206=1050.445,-111.019,432.591,169.952,30.544,155.797
C03207=1050.439,-111.269,432.600,169.949,30.543,155.797
C03208=1050.433,-111.519,432.610,169.947,30.543,155.797
C03209=1050.427,-111.769,432.620,169.946,30.542,155.797
C03210=1050.421,-112.018,432.629,169.944,30.542,155.797
C03211=1050.415,-112.268,432.639,169.941,30.541,155.797
C03212=1050.408,-112.517,432.649,169.939,30.540,155.797
C03213=1050.402,-112.767,432.659,169.937,30.540,155.797
C03214=1050.396,-113.017,432.668,169.935,30.540,155.797
C03215=1050.390,-113.267,432.678,169.933,30.539,155.797
C03216=1050.384,-113.517,432.688,169.930,30.539,155.797
C03217=1050.378,-113.767,432.697,169.928,30.538,155.797
C03218=1050.372,-114.016,432.707,169.926,30.538,155.797
C03219=1050.366,-114.266,432.717,169.924,30.537,155.797
C03220=1050.359,-114.516,432.726,169.921,30.537,155.798
C03221=1050.353,-114.766,432.736,169.919,30.537,155.798
C03222=1050.346,-115.051,432.746,169.918,30.536,155.798
C03223=1050.339,-115.336,432.757,169.915,30.536,155.798
C03224=1050.333,-115.621,432.768,169.913,30.535,155.798
C03225=1050.325,-115.906,432.779,169.910,30.534,155.798
C03226=1050.319,-116.156,432.788,169.908,30.534,155.798
C03227=1050.313,-116.406,432.798,169.906,30.534,155.798
C03228=1050.307,-116.655,432.808,169.903,30.533,155.798
C03229=1050.301,-116.905,432.817,169.901,30.533,155.798
C03230=1050.295,-117.155,432.827,169.899,30.533,155.798
C03231=1050.289,-117.404,432.836,169.897,30.532,155.798
C03232=1050.283,-117.654,432.845,169.894,30.532,155.798
C03233=1050.277,-117.904,432.855,169.892,30.531,155.798
C03234=1050.270,-118.153,432.864,169.890,30.531,155.799
C03235=1050.264,-118.403,432.874,169.888,30.531,155.799
C03236=1050.257,-118.653,432.883,169.886,30.530,155.799
C03237=1050.251,-118.903,432.893,169.884,30.530,155.799
C03238=1050.245,-119.153,432.902,169.882,30.530,155.799
C03239=1050.240,-119.402,432.911,169.880,30.529,155.799
C03240=1050.234,-119.652,432.920,169.877,30.529,155.799
C03241=1050.227,-119.902,432.930,169.875,30.528,155.799
C03242=1050.221,-120.151,432.939,169.873,30.528,155.799
C03243=1050.214,-120.401,432.948,169.871,30.528,155.799
C03244=1050.208,-120.651,432.958,169.869,30.527,155.799
C03245=1050.202,-120.901,432.967,169.866,30.527,155.799
C03246=1050.197,-121.150,432.976,169.864,30.527,155.799
C03247=1050.191,-121.400,432.986,169.862,30.526,155.800
C03248=1050.184,-121.650,432.995,169.860,30.526,155.800
C03249=1050.178,-121.900,433.005,169.857,30.526,155.800
C03250=1050.172,-122.150,433.013,169.856,30.525,155.800
C03251=1050.166,-122.399,433.022,169.854,30.525,155.800
C03252=1050.160,-122.649,433.032,169.852,30.525,155.800
C03253=1050.154,-122.898,433.041,169.849,30.525,155.800
C03254=1050.148,-123.149,433.050,169.847,30.524,155.800
C03255=1050.142,-123.399,433.060,169.845,30.524,155.800
C03256=1050.135,-123.647,433.068,169.843,30.524,155.800
C03257=1050.129,-123.897,433.078,169.840,30.523,155.800
C03258=1050.123,-124.148,433.087,169.838,30.523,155.800
C03259=1050.117,-124.397,433.096,169.836,30.523,155.801
C03260=1050.111,-124.647,433.106,169.834,30.523,155.801
C03261=1050.105,-124.897,433.114,169.831,30.522,155.801
C03262=1050.099,-125.146,433.123,169.829,30.522,155.801
C03263=1050.093,-125.396,433.133,169.827,30.522,155.801
C03264=1050.086,-125.646,433.141,169.825,30.522,155.801
C03265=1050.080,-125.895,433.150,169.822,30.522,155.801
C03266=1050.074,-126.145,433.160,169.821,30.521,155.801
C03267=1050.068,-126.396,433.169,169.819,30.521,155.801
C03268=1050.061,-126.645,433.178,169.817,30.521,155.802
C03269=1050.056,-126.894,433.187,169.814,30.521,155.802
C03270=1050.050,-127.145,433.196,169.812,30.520,155.802
C03271=1050.043,-127.394,433.205,169.810,30.520,155.802
C03272=1050.038,-127.643,433.214,169.808,30.520,155.802
C03273=1050.032,-127.894,433.223,169.805,30.520,155.802
C03274=1050.027,-128.143,433.233,169.803,30.519,155.802
C03275=1050.023,-128.393,433.243,169.801,30.518,155.802
C03276=1050.020,-128.643,433.255,169.799,30.516,155.802
C03277=1050.018,-128.893,433.266,169.798,30.514,155.801
C03278=1050.017,-129.144,433.279,169.797,30.512,155.801
C03279=1050.018,-129.394,433.291,169.795,30.508,155.801
C03280=1050.019,-129.645,433.305,169.793,30.504,155.800
C03281=1050.022,-129.894,433.318,169.793,30.500,155.799
C03282=1050.025,-130.145,433.333,169.792,30.496,155.799
C03283=1050.030,-130.396,433.350,169.790,30.490,155.798
C03284=1050.035,-130.647,433.366,169.790,30.485,155.797
C03285=1050.041,-130.896,433.382,169.789,30.479,155.796
C03286=1049.677,-130.920,433.156,169.743,30.648,155.828
C03287=1049.671,-130.671,433.140,169.744,30.654,155.829
C03288=1049.666,-130.420,433.123,169.745,30.660,155.830
C03289=1049.661,-130.169,433.108,169.746,30.665,155.831
C03290=1049.658,-129.918,433.093,169.747,30.670,155.832
C03291=1049.656,-129.668,433.078,169.748,30.674,155.832
C03292=1049.654,-129.418,433.065,169.749,30.677,155.833
C03293=1049.654,-129.167,433.052,169.751,30.681,155.833
C03294=1049.654,-128.917,433.039,169.753,30.683,155.834
C03295=1049.656,-128.667,433.028,169.753,30.685,155.834
C03296=1049.659,-128.417,433.017,169.755,30.687,155.834
C03297=1049.662,-128.167,433.006,169.757,30.689,155.834
C03298=1049.667,-127.917,432.997,169.759,30.689,155.834
C03299=1049.673,-127.667,432.987,169.762,30.689,155.834
C03300=1049.679,-127.418,432.978,169.764,30.690,155.834
C03301=1049.685,-127.168,432.970,169.766,30.690,155.834
C03302=1049.691,-126.918,432.960,169.768,30.690,155.834
C03303=1049.697,-126.669,432.951,169.771,30.690,155.834
C03304=1049.704,-126.419,432.943,169.773,30.690,155.834
C03305=1049.710,-126.169,432.933,169.775,30.691,155.833
C03306=1049.716,-125.919,432.923,169.778,30.691,155.833
C03307=1049.722,-125.670,432.916,169.780,30.691,155.833
C03308=1049.728,-125.420,432.906,169.781,30.691,155.833
C03309=1049.734,-125.170,432.896,169.783,30.692,155.833
C03310=1049.741,-124.920,432.888,169.786,30.692,155.833
C03311=1049.746,-124.671,432.879,169.788,30.692,155.833
C03312=1049.753,-124.421,432.869,169.790,30.692,155.833
C03313=1049.758,-124.171,432.861,169.792,30.692,155.833
C03314=1049.765,-123.921,432.851,169.795,30.693,155.833
C03315=1049.772,-123.671,432.842,169.797,30.693,155.832
C03316=1049.777,-123.422,432.833,169.799,30.693,155.832
C03317=1049.783,-123.172,432.824,169.801,30.693,155.832
C03318=1049.789,-122.922,432.814,169.804,30.694,155.832
C03319=1049.795,-122.672,432.805,169.806,30.694,155.832
C03320=1049.802,-122.423,432.796,169.808,30.694,155.832
C03321=1049.807,-122.173,432.787,169.810,30.695,155.832
C03322=1049.814,-121.923,432.778,169.813,30.695,155.832
C03323=1049.820,-121.673,432.768,169.815,30.695,155.832
C03324=1049.826,-121.424,432.759,169.817,30.695,155.832
C03325=1049.832,-121.173,432.750,169.818,30.695,155.832
C03326=1049.837,-120.924,432.741,169.821,30.696,155.831
C03327=1049.844,-120.675,432.732,169.823,30.696,155.831
C03328=1049.851,-120.425,432.722,169.825,30.697,155.831
C03329=1049.857,-120.175,432.713,169.827,30.697,155.831
C03330=1049.863,-119.925,432.703,169.830,30.697,155.831
C03331=1049.869,-119.675,432.694,169.832,30.698,155.831
C03332=1049.874,-119.426,432.685,169.834,30.698,155.831
C03333=1049.880,-119.176,432.675,169.836,30.698,155.831
C03334=1049.887,-118.926,432.666,169.839,30.699,155.831
C03335=1049.893,-118.676,432.656,169.841,30.699,155.831
C03336=1049.900,-118.427,432.647,169.843,30.699,155.831
C03337=1049.906,-118.177,432.638,169.845,30.700,155.831
C03338=1049.912,-117.927,432.628,169.848,30.700,155.831
C03339=1049.918,-117.678,432.619,169.849,30.700,155.830
C03340=1049.924,-117.427,432.610,169.851,30.701,155.830
C03341=1049.930,-117.178,432.600,169.853,30.701,155.830
C03342=1049.936,-116.928,432.591,169.856,30.702,155.830
C03343=1049.942,-116.678,432.581,169.858,30.702,155.830
C03344=1049.948,-116.429,432.572,169.860,30.702,155.830
C03345=1049.954,-116.179,432.562,169.862,30.703,155.830
C03346=1049.961,-115.929,432.553,169.865,30.703,155.830
C03347=1049.968,-115.644,432.542,169.867,30.703,155.830
C03348=1049.975,-115.359,432.531,169.870,30.704,155.830
C03349=1049.981,-115.074,432.520,169.872,30.704,155.830
C03350=1049.988,-114.789,432.510,169.875,30.705,155.830
C03351=1049.995,-114.539,432.500,169.877,30.706,155.830
C03352=1050.001,-114.289,432.490,169.879,30.706,155.830
C03353=1050.007,-114.039,432.481,169.881,30.706,155.830
C03354=1050.013,-113.790,432.471,169.883,30.707,155.829
C03355=1050.020,-113.541,432.461,169.885,30.707,155.829
C03356=1050.026,-113.291,432.451,169.887,30.707,155.829
C03357=1050.032,-113.041,432.442,169.889,30.708,155.829
C03358=1050.038,-112.791,432.432,169.892,30.709,155.829
C03359=1050.044,-112.541,432.423,169.894,30.709,155.829
C03360=1050.050,-112.291,432.413,169.896,30.709,155.829
C03361=1050.056,-112.041,432.403,169.898,30.710,155.829
C03362=1050.062,-111.792,432.393,169.901,30.711,155.829
C03363=1050.068,-111.542,432.384,169.903,30.711,155.829
C03364=1050.074,-111.292,432.374,169.905,30.711,155.829
C03365=1050.081,-111.043,432.364,169.907,30.712,155.829
C03366=1050.087,-110.793,432.354,169.909,30.713,155.829
C03367=1050.093,-110.543,432.345,169.911,30.713,155.829
C03368=1050.099,-110.293,432.335,169.913,30.713,155.829
C03369=1050.106,-110.044,432.326,169.915,30.714,155.829
C03370=1050.111,-109.794,432.316,169.917,30.715,155.829
C03371=1050.117,-109.544,432.305,169.920,30.715,155.829
C03372=1050.124,-109.295,432.296,169.922,30.715,155.829
C03373=1050.130,-109.045,432.286,169.924,30.716,155.828
C03374=1050.136,-108.795,432.277,169.926,30.717,155.829
C03375=1050.142,-108.545,432.267,169.928,30.717,155.828
C03376=1050.149,-108.296,432.257,169.931,30.717,155.828
C03377=1050.155,-108.046,432.247,169.933,30.718,155.828
C03378=1050.161,-107.796,432.238,169.935,30.719,155.828
C03379=1050.166,-107.546,432.227,169.937,30.719,155.828
C03380=1050.173,-107.297,432.217,169.939,30.720,155.828
C03381=1050.179,-107.047,432.208,169.941,30.720,155.828
C03382=1050.185,-106.798,432.198,169.943,30.721,155.828
C03383=1050.191,-106.548,432.187,169.945,30.721,155.828
C03384=1050.197,-106.298,432.178,169.947,30.722,155.828
C03385=1050.203,-106.048,432.168,169.950,30.722,155.828
C03386=1050.210,-105.798,432.158,169.952,30.723,155.828
C03387=1050.217,-105.549,432.148,169.954,30.724,155.828
C03388=1050.222,-105.299,432.138,169.956,30.725,155.828
C03389=1050.228,-105.049,432.128,169.959,30.725,155.828
C03390=1050.235,-104.800,432.118,169.961,30.725,155.828
C03391=1050.240,-104.550,432.108,169.963,30.726,155.828
C03392=1050.247,-104.300,432.097,169.964,30.727,155.828
C03393=1050.253,-104.051,432.088,169.966,30.728,155.828
C03394=1050.259,-103.801,432.078,169.969,30.728,155.828
C03395=1050.265,-103.551,432.067,169.971,30.729,155.828
C03396=1050.271,-103.301,432.058,169.973,30.729,155.828
C03397=1050.278,-103.052,432.047,169.975,30.730,155.828
C03398=1050.283,-102.801,432.037,169.977,30.731,155.828
C03399=1050.289,-102.552,432.027,169.980,30.732,155.828
C03400=1050.296,-102.303,432.017,169.982,30.732,155.828
C03401=1050.301,-102.052,432.007,169.984,30.733,155.828
C03402=1050.308,-101.803,431.997,169.986,30.733,155.828
C03403=1050.314,-101.553,431.987,169.988,30.734,155.828
C03404=1050.320,-101.304,431.976,169.990,30.735,155.828
C03405=1050.327,-101.053,431.966,169.992,30.736,155.828
C03406=1050.333,-100.804,431.956,169.994,30.736,155.828
C03407=1050.338,-100.554,431.946,169.996,30.737,155.828
C03408=1050.345,-100.305,431.936,169.999,30.737,155.828
C03409=1050.351,-100.055,431.926,170.001,30.738,155.828
C03410=1050.357,-99.806,431.915,170.003,30.739,155.828
C03411=1050.364,-99.518,431.904,170.005,30.740,155.828
C03412=1050.371,-99.232,431.892,170.008,30.741,155.828
C03413=1050.378,-98.946,431.881,170.010,30.741,155.828
C03414=1050.386,-98.660,431.869,170.013,30.742,155.828
C03415=1050.392,-98.410,431.858,170.014,30.743,155.828
C03416=1050.398,-98.160,431.848,170.016,30.743,155.828
C03417=1050.404,-97.911,431.838,170.019,30.744,155.828
C03418=1050.411,-97.661,431.827,170.021,30.745,155.828
C03419=1050.417,-97.411,431.817,170.023,30.746,155.828
C03420=1050.422,-97.162,431.806,170.025,30.747,155.828
C03421=1050.429,-96.912,431.797,170.027,30.748,155.828
C03422=1050.434,-96.662,431.786,170.030,30.748,155.828
C03423=1050.441,-96.413,431.775,170.032,30.749,155.828
C03424=1050.447,-96.162,431.765,170.034,30.750,155.828
C03425=1050.453,-95.913,431.754,170.036,30.751,155.828
C03426=1050.459,-95.664,431.744,170.037,30.751,155.828
C03427=1050.465,-95.414,431.734,170.039,30.752,155.828
C03428=1050.472,-95.164,431.723,170.042,30.753,155.828
C03429=1050.477,-94.914,431.712,170.044,30.754,155.828
C03430=1050.483,-94.664,431.702,170.046,30.754,155.828
C03431=1050.489,-94.415,431.692,170.048,30.755,155.828
C03432=1050.495,-94.166,431.681,170.050,30.756,155.828
C03433=1050.502,-93.916,431.670,170.053,30.757,155.828
C03434=1050.508,-93.666,431.660,170.055,30.758,155.828
C03435=1050.513,-93.416,431.649,170.057,30.759,155.828
C03436=1050.520,-93.167,431.639,170.058,30.760,155.828
C03437=1050.526,-92.917,431.628,170.060,30.760,155.828
C03438=1050.532,-92.667,431.618,170.062,30.761,155.828
C03439=1050.538,-92.417,431.607,170.065,30.763,155.828
C03440=1050.544,-92.168,431.596,170.067,30.763,155.828
C03441=1050.551,-91.918,431.586,170.069,30.764,155.828
C03442=1050.557,-91.669,431.575,170.071,30.765,155.828
C03443=1050.562,-91.418,431.565,170.073,30.766,155.828
C03444=1050.569,-91.169,431.554,170.075,30.767,155.828
C03445=1050.575,-90.919,431.543,170.078,30.768,155.828
C03446=1050.581,-90.670,431.533,170.079,30.769,155.828
C03447=1050.587,-90.420,431.522,170.081,30.770,155.828
C03448=1050.593,-90.170,431.511,170.083,30.770,155.828
C03449=1050.600,-89.920,431.501,170.085,30.771,155.828
C03450=1050.605,-89.671,431.490,170.088,30.772,155.828
C03451=1050.612,-89.421,431.479,170.090,30.773,155.828
C03452=1050.618,-89.172,431.469,170.092,30.774,155.828
C03453=1050.624,-88.922,431.458,170.094,30.775,155.828
C03454=1050.630,-88.672,431.447,170.096,30.776,155.828
C03455=1050.637,-88.423,431.436,170.098,30.777,155.828
C03456=1050.642,-88.173,431.426,170.100,30.778,155.828
C03457=1050.648,-87.922,431.415,170.102,30.779,155.828
C03458=1050.655,-87.673,431.405,170.104,30.779,155.829
C03459=1050.661,-87.423,431.393,170.106,30.780,155.829
C03460=1050.667,-87.174,431.383,170.108,30.781,155.828
C03461=1050.673,-86.924,431.372,170.110,30.782,155.829
C03462=1050.680,-86.674,431.361,170.113,30.783,155.829
C03463=1050.686,-86.425,431.350,170.115,30.784,155.829
C03464=1050.693,-86.175,431.340,170.117,30.785,155.829
C03465=1050.698,-85.925,431.329,170.119,30.786,155.829
C03466=1050.704,-85.676,431.318,170.121,30.786,155.829
C03467=1050.711,-85.426,431.307,170.122,30.787,155.829
C03468=1050.717,-85.176,431.296,170.124,30.788,155.829
C03469=1050.723,-84.926,431.285,170.127,30.789,155.829
C03470=1050.730,-84.677,431.275,170.129,30.790,155.829
C03471=1050.735,-84.428,431.264,170.131,30.791,155.829
C03472=1050.742,-84.177,431.253,170.133,30.792,155.829
C03473=1050.748,-83.928,431.242,170.135,30.793,155.829
C03474=1050.755,-83.678,431.231,170.137,30.794,155.829
C03475=1050.762,-83.394,431.218,170.140,30.795,155.829
C03476=1050.769,-83.110,431.206,170.142,30.796,155.829
C03477=1050.776,-82.826,431.193,170.144,30.797,155.829
C03478=1050.783,-82.542,431.180,170.146,30.799,155.829
C03479=1050.789,-82.293,431.170,170.148,30.800,155.829
C03480=1050.796,-82.043,431.159,170.151,30.801,155.829
C03481=1050.801,-81.793,431.148,170.153,30.802,155.829
C03482=1050.808,-81.543,431.137,170.155,30.803,155.829
C03483=1050.814,-81.294,431.127,170.157,30.804,155.830
C03484=1050.821,-81.044,431.115,170.159,30.804,155.830
C03485=1050.827,-80.795,431.104,170.161,30.805,155.830
C03486=1050.834,-80.545,431.093,170.163,30.807,155.830
C03487=1050.839,-80.295,431.082,170.165,30.807,155.830
C03488=1050.846,-80.045,431.071,170.167,30.808,155.830
C03489=1050.851,-79.796,431.060,170.169,30.809,155.830
C03490=1050.858,-79.546,431.048,170.171,30.810,155.830
C03491=1050.864,-79.297,431.037,170.173,30.811,155.830
C03492=1050.871,-79.047,431.027,170.175,30.813,155.830
C03493=1050.877,-78.797,431.016,170.177,30.814,155.830
C03494=1050.883,-78.547,431.004,170.180,30.815,155.830
C03495=1050.889,-78.298,430.993,170.181,30.816,155.830
C03496=1050.895,-78.048,430.982,170.183,30.817,155.830
C03497=1050.901,-77.798,430.971,170.185,30.818,155.830
C03498=1050.908,-77.549,430.959,170.187,30.819,155.830
C03499=1050.913,-77.299,430.948,170.189,30.820,155.830
C03500=1050.920,-77.049,430.937,170.191,30.822,155.831
C03501=1050.926,-76.800,430.926,170.194,30.823,155.831
C03502=1050.932,-76.550,430.914,170.196,30.824,155.831
C03503=1050.938,-76.301,430.903,170.198,30.824,155.831
C03504=1050.944,-76.050,430.892,170.199,30.826,155.831
C03505=1050.951,-75.801,430.880,170.201,30.827,155.831
C03506=1050.957,-75.551,430.869,170.203,30.828,155.831
C03507=1050.963,-75.301,430.858,170.205,30.829,155.831
C03508=1050.969,-75.052,430.846,170.207,30.830,155.831
C03509=1050.975,-74.802,430.835,170.210,30.831,155.831
C03510=1050.981,-74.553,430.824,170.212,30.832,155.831
C03511=1050.988,-74.303,430.812,170.214,30.833,155.831
C03512=1050.994,-74.053,430.801,170.216,30.835,155.831
C03513=1051.000,-73.804,430.789,170.218,30.836,155.832
C03514=1051.007,-73.554,430.778,170.219,30.837,155.832
C03515=1051.013,-73.305,430.766,170.221,30.838,155.832
C03516=1051.018,-73.054,430.754,170.223,30.840,155.832
C03517=1051.024,-72.805,430.744,170.225,30.841,155.832
C03518=1051.031,-72.555,430.732,170.228,30.842,155.832
C03519=1051.036,-72.306,430.721,170.230,30.843,155.832
C03520=1051.042,-72.056,430.708,170.232,30.844,155.832
C03521=1051.048,-71.807,430.697,170.234,30.846,155.832
C03522=1051.055,-71.557,430.685,170.235,30.847,155.832
C03523=1051.061,-71.307,430.674,170.237,30.848,155.833
C03524=1051.066,-71.058,430.662,170.239,30.849,155.833
C03525=1051.073,-70.807,430.651,170.241,30.851,155.833
C03526=1051.079,-70.559,430.639,170.243,30.852,155.833
C03527=1051.085,-70.308,430.628,170.245,30.853,155.833
C03528=1051.091,-70.058,430.615,170.247,30.854,155.833
C03529=1051.097,-69.810,430.604,170.250,30.856,155.833
C03530=1051.103,-69.559,430.592,170.252,30.857,155.833
C03531=1051.109,-69.311,430.581,170.253,30.858,155.833
C03532=1051.115,-69.060,430.569,170.255,30.859,155.833
C03533=1051.122,-68.810,430.557,170.257,30.861,155.834
C03534=1051.127,-68.561,430.546,170.259,30.862,155.834
C03535=1051.134,-68.311,430.534,170.261,30.863,155.834
C03536=1051.140,-68.062,430.522,170.263,30.864,155.834
C03537=1051.146,-67.812,430.511,170.265,30.866,155.834
C03538=1051.152,-67.562,430.499,170.267,30.867,155.834
C03539=1051.159,-67.281,430.485,170.269,30.868,155.834
C03540=1051.165,-66.998,430.472,170.271,30.870,155.834
C03541=1051.172,-66.716,430.459,170.273,30.871,155.834
C03542=1051.180,-66.435,430.446,170.276,30.873,155.835
C03543=1051.186,-66.185,430.433,170.278,30.874,155.835
C03544=1051.192,-65.935,430.422,170.280,30.876,155.835
C03545=1051.198,-65.686,430.411,170.282,30.877,155.835
C03546=1051.205,-65.437,430.399,170.284,30.878,155.835
C03547=1051.210,-65.186,430.387,170.286,30.879,155.835
C03548=1051.217,-64.937,430.375,170.287,30.881,155.835
C03549=1051.223,-64.688,430.363,170.289,30.882,155.835
C03550=1051.228,-64.437,430.351,170.291,30.883,155.835
C03551=1051.235,-64.188,430.339,170.294,30.885,155.836
C03552=1051.241,-63.939,430.328,170.296,30.886,155.836
C03553=1051.247,-63.689,430.315,170.298,30.887,155.836
C03554=1051.253,-63.439,430.304,170.300,30.889,155.836
C03555=1051.260,-63.189,430.292,170.302,30.890,155.836
C03556=1051.265,-62.940,430.280,170.303,30.891,155.836
C03557=1051.272,-62.691,430.268,170.305,30.892,155.836
C03558=1051.279,-62.441,430.256,170.307,30.894,155.836
C03559=1051.284,-62.190,430.244,170.309,30.895,155.837
C03560=1051.290,-61.942,430.233,170.311,30.896,155.837
C03561=1051.297,-61.692,430.221,170.313,30.898,155.837
C03562=1051.303,-61.442,430.208,170.315,30.899,155.837
C03563=1051.310,-61.193,430.196,170.317,30.900,155.837
C03564=1051.316,-60.942,430.185,170.319,30.902,155.837
C03565=1051.321,-60.693,430.173,170.321,30.903,155.837
C03566=1051.328,-60.444,430.161,170.323,30.904,155.837
C03567=1051.334,-60.194,430.149,170.325,30.906,155.837
C03568=1051.340,-59.944,430.136,170.327,30.907,155.838
C03569=1051.347,-59.695,430.124,170.329,30.908,155.838
C03570=1051.353,-59.446,430.113,170.331,30.910,155.838
C03571=1051.359,-59.196,430.100,170.333,30.911,155.838
C03572=1051.365,-58.946,430.089,170.335,30.912,155.838
C03573=1051.372,-58.696,430.077,170.336,30.914,155.838
C03574=1051.378,-58.446,430.064,170.338,30.915,155.838
C03575=1051.385,-58.197,430.052,170.340,30.916,155.838
C03576=1051.391,-57.948,430.041,170.342,30.918,155.839
C03577=1051.396,-57.698,430.028,170.344,30.919,155.839
C03578=1051.403,-57.448,430.016,170.346,30.920,155.839
C03579=1051.409,-57.198,430.004,170.349,30.922,155.839
C03580=1051.416,-56.949,429.992,170.351,30.923,155.839
C03581=1051.422,-56.699,429.980,170.352,30.924,155.839
C03582=1051.428,-56.449,429.967,170.354,30.926,155.839
C03583=1051.435,-56.200,429.955,170.356,30.927,155.839
C03584=1051.441,-55.950,429.943,170.358,30.928,155.840
C03585=1051.447,-55.701,429.931,170.360,30.930,155.840
C03586=1051.453,-55.452,429.919,170.362,30.932,155.840
C03587=1051.459,-55.202,429.907,170.364,30.932,155.840
C03588=1051.466,-54.952,429.895,170.366,30.934,155.840
C03589=1051.473,-54.702,429.883,170.368,30.936,155.840
C03590=1051.479,-54.453,429.870,170.369,30.936,155.840
C03591=1051.485,-54.203,429.858,170.371,30.938,155.840
C03592=1051.491,-53.953,429.846,170.373,30.940,155.841
C03593=1051.498,-53.704,429.834,170.375,30.941,155.841
C03594=1051.504,-53.454,429.821,170.377,30.942,155.841
C03595=1051.510,-53.204,429.809,170.379,30.944,155.841
C03596=1051.517,-52.955,429.797,170.381,30.945,155.841
C03597=1051.523,-52.705,429.784,170.383,30.947,155.841
C03598=1051.530,-52.456,429.772,170.385,30.948,155.841
C03599=1051.536,-52.206,429.759,170.387,30.949,155.842
C03600=1051.542,-51.956,429.747,170.389,30.951,155.842
C03601=1051.549,-51.707,429.736,170.391,30.952,155.842
C03602=1051.555,-51.457,429.723,170.393,30.953,155.842
C03603=1051.562,-51.176,429.709,170.395,30.955,155.842
C03604=1051.569,-50.896,429.695,170.397,30.956,155.842
C03605=1051.576,-50.615,429.681,170.400,30.958,155.842
C03606=1051.583,-50.335,429.668,170.401,30.959,155.843
C03607=1051.590,-50.085,429.655,170.403,30.961,155.843
C03608=1051.596,-49.835,429.642,170.405,30.963,155.843
C03609=1051.602,-49.586,429.630,170.407,30.964,155.843
C03610=1051.608,-49.336,429.618,170.409,30.966,155.843
C03611=1051.614,-49.087,429.605,170.411,30.967,155.843
C03612=1051.620,-48.838,429.592,170.413,30.969,155.843
C03613=1051.626,-48.588,429.580,170.415,30.970,155.844
C03614=1051.632,-48.338,429.568,170.416,30.972,155.844
C03615=1051.638,-48.089,429.554,170.418,30.973,155.844
C03616=1051.644,-47.839,429.542,170.420,30.975,155.844
C03617=1051.651,-47.589,429.530,170.422,30.976,155.844
C03618=1051.657,-47.340,429.517,170.424,30.978,155.844
C03619=1051.663,-47.090,429.504,170.426,30.979,155.845
C03620=1051.669,-46.840,429.491,170.428,30.981,155.845
C03621=1051.676,-46.591,429.479,170.430,30.982,155.845
C03622=1051.682,-46.342,429.466,170.431,30.984,155.845
C03623=1051.688,-46.092,429.454,170.433,30.986,155.845
C03624=1051.694,-45.842,429.440,170.435,30.987,155.845
C03625=1051.701,-45.593,429.428,170.437,30.989,155.846
C03626=1051.707,-45.343,429.416,170.439,30.990,155.846
C03627=1051.713,-45.094,429.403,170.441,30.992,155.846
C03628=1051.719,-44.844,429.390,170.443,30.993,155.846
C03629=1051.725,-44.594,429.377,170.445,30.995,155.846
C03630=1051.732,-44.345,429.365,170.446,30.996,155.846
C03631=1051.737,-44.095,429.352,170.448,30.998,155.847
